C03630=1074.416,86.468,-68.167,173.484,24.240,154.290
C03631=1074.422,86.718,-68.185,173.486,24.243,154.290
C03632=1074.428,86.966,-68.204,173.487,24.245,154.290
C03633=1074.434,87.216,-68.222,173.489,24.248,154.290
C03634=1074.440,87.465,-68.239,173.491,24.251,154.291
C03635=1074.446,87.715,-68.257,173.492,24.253,154.291
C03636=1074.451,87.964,-68.275,173.493,24.256,154.291
C03637=1074.458,88.213,-68.293,173.496,24.259,154.292
C03638=1074.463,88.462,-68.311,173.497,24.261,154.292
C03639=1074.469,88.712,-68.329,173.498,24.263,154.292
C03640=1074.475,88.961,-68.346,173.500,24.266,154.293
C03641=1074.481,89.210,-68.366,173.502,24.269,154.293
C03642=1074.486,89.459,-68.383,173.503,24.271,154.293
C03643=1074.492,89.709,-68.401,173.504,24.274,154.294
C03644=1074.498,89.958,-68.419,173.506,24.276,154.294
C03645=1074.504,90.207,-68.437,173.508,24.279,154.294
C03646=1074.510,90.457,-68.455,173.509,24.282,154.294
C03647=1074.516,90.706,-68.473,173.511,24.284,154.295
C03648=1074.522,90.955,-68.491,173.512,24.286,154.295
C03649=1074.527,91.204,-68.510,173.514,24.289,154.295
C03650=1074.533,91.454,-68.528,173.516,24.292,154.296
C03651=1074.539,91.702,-68.546,173.517,24.294,154.296
C03652=1074.544,91.952,-68.564,173.519,24.297,154.296
C03653=1074.550,92.201,-68.582,173.521,24.299,154.297
C03654=1074.556,92.451,-68.601,173.522,24.302,154.297
C03655=1074.561,92.700,-68.619,173.523,24.305,154.297
C03656=1074.567,92.950,-68.637,173.525,24.307,154.298
C03657=1074.573,93.198,-68.655,173.527,24.310,154.298
C03658=1074.578,93.448,-68.673,173.528,24.313,154.298
C03659=1074.584,93.697,-68.692,173.529,24.315,154.299
C03660=1074.590,93.946,-68.710,173.532,24.318,154.299
C03661=1074.595,94.196,-68.728,173.533,24.321,154.299
C03662=1074.602,94.445,-68.747,173.534,24.323,154.299
C03663=1074.608,94.727,-68.768,173.536,24.326,154.300
C03664=1074.614,95.008,-68.788,173.538,24.329,154.300
C03665=1074.621,95.290,-68.808,173.540,24.332,154.301
C03666=1074.627,95.571,-68.829,173.541,24.334,154.301
C03667=1074.633,95.820,-68.848,173.543,24.337,154.301
C03668=1074.639,96.070,-68.866,173.545,24.340,154.301
C03669=1074.644,96.319,-68.884,173.546,24.342,154.302
C03670=1074.651,96.568,-68.902,173.547,24.344,154.302
C03671=1074.656,96.817,-68.921,173.549,24.348,154.302
C03672=1074.662,97.067,-68.939,173.551,24.350,154.303
C03673=1074.668,97.316,-68.958,173.552,24.352,154.303
C03674=1074.673,97.565,-68.976,173.555,24.355,154.303
C03675=1074.679,97.814,-68.995,173.556,24.358,154.304
C03676=1074.684,98.064,-69.013,173.557,24.360,154.304
C03677=1074.691,98.313,-69.031,173.558,24.363,154.304
C03678=1074.697,98.563,-69.049,173.561,24.365,154.304
C03679=1074.702,98.811,-69.068,173.562,24.368,154.305
C03680=1074.708,99.061,-69.087,173.563,24.370,154.305
C03681=1074.714,99.311,-69.105,173.566,24.373,154.305
C03682=1074.719,99.559,-69.124,173.567,24.376,154.306
C03683=1074.726,99.809,-69.142,173.568,24.378,154.306
C03684=1074.731,100.058,-69.161,173.570,24.381,154.306
C03685=1074.737,100.307,-69.179,173.572,24.383,154.307
C03686=1074.742,100.557,-69.198,173.573,24.386,154.307
C03687=1074.749,100.806,-69.216,173.575,24.388,154.307
C03688=1074.754,101.055,-69.235,173.577,24.391,154.308
C03689=1074.760,101.304,-69.253,173.578,24.394,154.308
C03690=1074.766,101.554,-69.272,173.580,24.396,154.308
C03691=1074.772,101.802,-69.291,173.581,24.398,154.308
C03692=1074.777,102.052,-69.309,173.583,24.401,154.309
C03693=1074.783,102.301,-69.327,173.584,24.404,154.309
C03694=1074.788,102.550,-69.347,173.586,24.406,154.309
C03695=1074.794,102.800,-69.365,173.588,24.409,154.310
C03696=1074.800,103.049,-69.384,173.589,24.412,154.310
C03697=1074.805,103.298,-69.403,173.591,24.414,154.310
C03698=1074.811,103.547,-69.422,173.593,24.417,154.311
C03699=1074.817,103.796,-69.440,173.594,24.419,154.311
C03700=1074.822,104.046,-69.459,173.596,24.422,154.311
C03701=1074.829,104.295,-69.477,173.597,24.424,154.312
C03702=1074.834,104.544,-69.496,173.599,24.427,154.312
C03703=1074.839,104.793,-69.516,173.601,24.429,154.312
C03704=1074.846,105.043,-69.534,173.602,24.432,154.312
C03705=1074.851,105.292,-69.552,173.604,24.435,154.313
C03706=1074.856,105.541,-69.572,173.606,24.437,154.313
C03707=1074.863,105.790,-69.590,173.607,24.440,154.313
C03708=1074.868,106.040,-69.610,173.609,24.442,154.314
C03709=1074.873,106.289,-69.628,173.611,24.445,154.314
C03710=1074.880,106.538,-69.646,173.612,24.447,154.314
C03711=1074.885,106.788,-69.666,173.614,24.450,154.315
C03712=1074.890,107.036,-69.684,173.615,24.453,154.315
C03713=1074.897,107.285,-69.703,173.617,24.455,154.315
C03714=1074.903,107.535,-69.722,173.618,24.457,154.315
C03715=1074.908,107.784,-69.742,173.620,24.460,154.316
C03716=1074.914,108.033,-69.760,173.622,24.463,154.316
C03717=1074.919,108.283,-69.778,173.623,24.465,154.316
C03718=1074.925,108.532,-69.798,173.625,24.468,154.317
C03719=1074.932,108.781,-69.816,173.627,24.470,154.317
C03720=1074.937,109.030,-69.835,173.628,24.473,154.317
C03721=1074.942,109.279,-69.854,173.630,24.476,154.317
C03722=1074.948,109.529,-69.874,173.632,24.478,154.318
C03723=1074.954,109.778,-69.892,173.633,24.480,154.318
C03724=1074.960,110.027,-69.912,173.635,24.483,154.318
C03725=1074.965,110.276,-69.930,173.637,24.486,154.319
C03726=1074.972,110.525,-69.949,173.638,24.488,154.319
C03727=1074.978,110.807,-69.971,173.640,24.491,154.319
C03728=1074.985,111.089,-69.992,173.642,24.494,154.320
C03729=1074.991,111.370,-70.014,173.644,24.496,154.320
C03730=1074.998,111.652,-70.036,173.646,24.500,154.320
C03731=1075.003,111.901,-70.055,173.647,24.502,154.321
C03732=1075.009,112.151,-70.074,173.650,24.505,154.321
C03733=1075.015,112.400,-70.093,173.651,24.507,154.321
C03734=1075.020,112.648,-70.112,173.652,24.509,154.321
C03735=1075.026,112.898,-70.131,173.655,24.513,154.322
C03736=1075.032,113.147,-70.150,173.656,24.515,154.322
C03737=1075.037,113.397,-70.169,173.657,24.517,154.322
C03738=1075.043,113.646,-70.189,173.660,24.520,154.323
C03739=1075.048,113.895,-70.207,173.661,24.522,154.323
C03740=1075.055,114.144,-70.226,173.662,24.525,154.323
C03741=1075.061,114.393,-70.246,173.665,24.527,154.323
C03742=1075.066,114.642,-70.265,173.666,24.530,154.324
C03743=1075.072,114.892,-70.285,173.667,24.533,154.324
C03744=1075.077,115.140,-70.303,173.670,24.535,154.324
C03745=1075.083,115.390,-70.323,173.671,24.538,154.325
C03746=1075.089,115.639,-70.342,173.672,24.541,154.325
C03747=1075.095,115.888,-70.362,173.675,24.543,154.325
C03748=1075.099,116.138,-70.382,173.676,24.546,154.326
C03749=1075.105,116.387,-70.401,173.677,24.548,154.326
C03750=1075.110,116.636,-70.420,173.680,24.551,154.326
C03751=1075.116,116.885,-70.439,173.681,24.554,154.327
C03752=1075.122,117.134,-70.459,173.682,24.556,154.327
C03753=1075.128,117.384,-70.478,173.684,24.559,154.327
C03754=1075.133,117.633,-70.498,173.686,24.561,154.327
C03755=1075.138,117.882,-70.516,173.687,24.563,154.328
C03756=1075.144,118.131,-70.536,173.689,24.566,154.328
C03757=1075.150,118.380,-70.556,173.691,24.569,154.328
C03758=1075.156,118.630,-70.575,173.693,24.572,154.329
C03759=1075.162,118.878,-70.595,173.694,24.574,154.329
C03760=1075.167,119.128,-70.614,173.696,24.576,154.329
C03761=1075.173,119.377,-70.633,173.698,24.579,154.330
C03762=1075.177,119.626,-70.653,173.699,24.582,154.330
C03763=1075.183,119.875,-70.673,173.701,24.584,154.330
C03764=1075.189,120.125,-70.692,173.703,24.587,154.330
C03765=1075.195,120.374,-70.711,173.704,24.589,154.331
C03766=1075.201,120.623,-70.731,173.707,24.592,154.331
C03767=1075.207,120.872,-70.750,173.708,24.594,154.331
C03768=1075.213,121.121,-70.770,173.710,24.597,154.332
C03769=1075.218,121.370,-70.790,173.712,24.600,154.332
C03770=1075.224,121.620,-70.809,173.713,24.602,154.332
C03771=1075.229,121.869,-70.829,173.714,24.604,154.333
C03772=1075.234,122.118,-70.848,173.717,24.607,154.333
C03773=1075.240,122.367,-70.868,173.718,24.609,154.333
C03774=1075.246,122.616,-70.887,173.720,24.612,154.333
C03775=1075.252,122.865,-70.907,173.722,24.614,154.334
C03776=1075.258,123.114,-70.927,173.723,24.617,154.334
C03777=1075.263,123.364,-70.946,173.726,24.619,154.334
C03778=1075.269,123.613,-70.966,173.727,24.622,154.335
C03779=1075.274,123.862,-70.986,173.728,24.625,154.335
C03780=1075.280,124.111,-71.006,173.730,24.627,154.335
C03781=1075.286,124.360,-71.025,173.732,24.630,154.335
C03782=1075.292,124.609,-71.045,173.734,24.632,154.336
C03783=1075.298,124.859,-71.064,173.736,24.635,154.336
C03784=1075.304,125.108,-71.084,173.737,24.637,154.336
C03785=1075.309,125.357,-71.104,173.739,24.640,154.337
C03786=1075.315,125.606,-71.124,173.741,24.642,154.337
C03787=1075.320,125.856,-71.143,173.743,24.645,154.337
C03788=1075.326,126.104,-71.163,173.744,24.647,154.337
C03789=1075.332,126.354,-71.182,173.746,24.649,154.338
C03790=1075.337,126.603,-71.203,173.748,24.652,154.338
C03791=1075.344,126.885,-71.225,173.750,24.655,154.338
C03792=1075.351,127.166,-71.247,173.752,24.658,154.339
C03793=1075.357,127.448,-71.270,173.754,24.661,154.339
C03794=1075.364,127.729,-71.292,173.756,24.664,154.339
C03795=1075.370,127.978,-71.312,173.757,24.666,154.340
C03796=1075.374,128.228,-71.332,173.760,24.669,154.340
C03797=1075.380,128.477,-71.352,173.761,24.671,154.340
C03798=1075.386,128.725,-71.371,173.762,24.673,154.340
C03799=1075.392,128.975,-71.391,173.765,24.676,154.341
C03800=1075.399,129.224,-71.411,173.766,24.678,154.341
C03801=1075.404,129.473,-71.432,173.768,24.681,154.341
C03802=1075.410,129.723,-71.451,173.770,24.683,154.341
C03803=1075.416,129.972,-71.471,173.771,24.686,154.342
C03804=1075.422,130.220,-71.491,173.774,24.688,154.342
C03805=1075.427,130.470,-71.511,173.775,24.691,154.342
C03806=1075.433,130.719,-71.531,173.777,24.693,154.343
C03807=1075.439,130.968,-71.551,173.779,24.696,154.343
C03808=1075.445,131.217,-71.570,173.781,24.698,154.343
C03809=1075.450,131.466,-71.590,173.782,24.701,154.343
C03810=1075.456,131.716,-71.611,173.784,24.703,154.344
C03811=1075.462,131.965,-71.631,173.786,24.706,154.344
C03812=1075.468,132.214,-71.651,173.787,24.708,154.344
C03813=1075.473,132.463,-71.671,173.790,24.711,154.345
C03814=1075.479,132.712,-71.690,173.791,24.713,154.345
C03815=1075.484,132.961,-71.711,173.793,24.716,154.345
C03816=1075.490,133.210,-71.731,173.795,24.718,154.345
C03817=1075.496,133.459,-71.751,173.796,24.720,154.346
C03818=1075.502,133.708,-71.771,173.799,24.723,154.346
C03819=1075.507,133.958,-71.791,173.800,24.725,154.346
C03820=1075.513,134.207,-71.811,173.802,24.729,154.347
C03821=1075.518,134.456,-71.832,173.804,24.731,154.347
C03822=1075.524,134.705,-71.852,173.806,24.734,154.347
C03823=1075.530,134.954,-71.873,173.807,24.736,154.347
C03824=1075.536,135.203,-71.893,173.810,24.739,154.348
C03825=1075.541,135.452,-71.913,173.811,24.741,154.348
C03826=1075.547,135.701,-71.933,173.812,24.743,154.348
C03827=1075.552,135.950,-71.954,173.815,24.746,154.349
C03828=1075.558,136.200,-71.973,173.816,24.748,154.349
C03829=1075.564,136.449,-71.994,173.818,24.751,154.349
C03830=1075.570,136.698,-72.014,173.820,24.753,154.349
C03831=1075.575,136.947,-72.034,173.822,24.756,154.350
C03832=1075.581,137.196,-72.054,173.823,24.758,154.350
C03833=1075.586,137.445,-72.075,173.826,24.761,154.350
C03834=1075.592,137.694,-72.095,173.827,24.763,154.350
C03835=1075.598,137.944,-72.116,173.829,24.766,154.351
C03836=1075.604,138.193,-72.136,173.831,24.768,154.351
C03837=1075.609,138.442,-72.156,173.832,24.771,154.351
C03838=1075.615,138.691,-72.176,173.835,24.773,154.352
C03839=1075.621,138.940,-72.197,173.836,24.776,154.352
C03840=1075.626,139.189,-72.217,173.838,24.778,154.352
C03841=1075.632,139.438,-72.238,173.840,24.781,154.352
C03842=1075.638,139.688,-72.258,173.842,24.783,154.353
C03843=1075.644,139.936,-72.278,173.843,24.786,154.353
C03844=1075.649,140.185,-72.299,173.846,24.788,154.353
C03845=1075.654,140.434,-72.320,173.847,24.791,154.353
C03846=1075.661,140.684,-72.340,173.849,24.793,154.354
C03847=1075.666,140.933,-72.361,173.851,24.796,154.354
C03848=1075.672,141.182,-72.381,173.853,24.798,154.354
C03849=1075.678,141.431,-72.401,173.855,24.801,154.355
C03850=1075.683,141.680,-72.422,173.857,24.803,154.355
C03851=1075.689,141.930,-72.443,173.858,24.806,154.355
C03852=1075.694,142.178,-72.464,173.861,24.808,154.355
C03853=1075.700,142.427,-72.484,173.862,24.811,154.356
C03854=1075.705,142.676,-72.505,173.864,24.813,154.356
C03855=1075.712,142.958,-72.528,173.866,24.816,154.356
C03856=1075.719,143.239,-72.551,173.868,24.819,154.357
C03857=1075.725,143.520,-72.574,173.870,24.822,154.357
C03858=1075.731,143.802,-72.598,173.872,24.825,154.357
C03859=1075.736,144.051,-72.618,173.874,24.827,154.358
C03860=1075.742,144.301,-72.639,173.876,24.830,154.358
C03861=1075.748,144.549,-72.661,173.878,24.832,154.358
C03862=1075.754,144.798,-72.680,173.880,24.835,154.358
C03863=1075.759,145.047,-72.701,173.881,24.837,154.359
C03864=1075.765,145.297,-72.722,173.884,24.840,154.359
C03865=1075.770,145.546,-72.743,173.885,24.842,154.359
C03866=1075.776,145.795,-72.763,173.887,24.845,154.359
C03867=1075.782,146.044,-72.784,173.889,24.847,154.360
C03868=1075.788,146.293,-72.805,173.891,24.850,154.360
C03869=1075.793,146.542,-72.826,173.892,24.852,154.360
C03870=1075.799,146.791,-72.846,173.895,24.855,154.361
C03871=1075.805,147.040,-72.868,173.896,24.857,154.361
C03872=1075.811,147.289,-72.888,173.898,24.860,154.361
C03873=1075.816,147.538,-72.909,173.900,24.862,154.361
C03874=1075.822,147.787,-72.930,173.902,24.865,154.362
C03875=1075.828,148.036,-72.950,173.904,24.867,154.362
C03876=1075.833,148.285,-72.971,173.906,24.870,154.362
C03877=1075.839,148.535,-72.992,173.908,24.872,154.362
C03878=1075.845,148.784,-73.013,173.910,24.875,154.363
C03879=1075.850,149.032,-73.034,173.912,24.877,154.363
C03880=1075.856,149.282,-73.055,173.913,24.880,154.363
C03881=1075.862,149.531,-73.076,173.916,24.882,154.364
C03882=1075.867,149.780,-73.097,173.917,24.885,154.364
C03883=1075.873,150.030,-73.118,173.919,24.887,154.364
C03884=1075.878,150.278,-73.139,173.921,24.890,154.364
C03885=1075.884,150.527,-73.160,173.923,24.892,154.365
C03886=1075.890,150.776,-73.181,173.925,24.895,154.365
C03887=1075.895,151.025,-73.202,173.927,24.897,154.365
C03888=1075.901,151.274,-73.223,173.928,24.899,154.366
C03889=1075.906,151.524,-73.244,173.931,24.902,154.366
C03890=1075.912,151.772,-73.265,173.932,24.904,154.366
C03891=1075.917,152.021,-73.286,173.934,24.907,154.366
C03892=1075.923,152.271,-73.308,173.937,24.910,154.367
C03893=1075.929,152.519,-73.329,173.938,24.912,154.367
C03894=1075.935,152.769,-73.350,173.940,24.915,154.367
C03895=1075.940,153.017,-73.371,173.942,24.917,154.367
C03896=1075.946,153.267,-73.392,173.944,24.920,154.368
C03897=1075.952,153.516,-73.413,173.946,24.922,154.368
C03898=1075.957,153.765,-73.434,173.948,24.924,154.368
C03899=1075.963,154.013,-73.455,173.949,24.926,154.368
C03900=1075.969,154.263,-73.477,173.952,24.929,154.369
C03901=1075.974,154.512,-73.497,173.954,24.932,154.369
C03902=1075.980,154.761,-73.519,173.956,24.934,154.369
C03903=1075.986,155.009,-73.540,173.958,24.937,154.369
C03904=1075.992,155.259,-73.561,173.959,24.939,154.370
C03905=1075.997,155.508,-73.582,173.962,24.942,154.370
C03906=1076.003,155.756,-73.604,173.963,24.944,154.370
C03907=1076.009,156.006,-73.625,173.965,24.947,154.371
C03908=1076.013,156.255,-73.646,173.968,24.949,154.371
C03909=1076.020,156.504,-73.668,173.969,24.952,154.371
C03910=1076.025,156.753,-73.689,173.971,24.954,154.371
C03911=1076.031,157.002,-73.710,173.973,24.957,154.372
C03912=1076.037,157.251,-73.731,173.975,24.959,154.372
C03913=1076.042,157.499,-73.753,173.977,24.962,154.372
C03914=1076.047,157.750,-73.774,173.979,24.964,154.373
C03915=1076.053,157.998,-73.796,173.981,24.967,154.373
C03916=1076.059,158.247,-73.817,173.983,24.969,154.373
C03917=1076.064,158.496,-73.838,173.985,24.972,154.373
C03918=1076.071,158.745,-73.860,173.986,24.974,154.374
C03919=1076.076,159.027,-73.884,173.989,24.977,154.374
C03920=1076.083,159.307,-73.908,173.991,24.980,154.374
C03921=1076.089,159.589,-73.932,173.993,24.983,154.375
C03922=1076.096,159.870,-73.957,173.996,24.985,154.375
C03923=1076.102,160.119,-73.978,173.998,24.988,154.375
C03924=1076.107,160.368,-74.000,173.999,24.990,154.375
C03925=1076.113,160.618,-74.021,174.002,24.993,154.376
C03926=1076.118,160.866,-74.042,174.003,24.995,154.376
C03927=1076.124,161.115,-74.064,174.005,24.998,154.376
C03928=1076.129,161.364,-74.086,174.008,25.001,154.376
C03929=1076.135,161.613,-74.107,174.009,25.003,154.377
C03930=1076.141,161.862,-74.129,174.011,25.006,154.377
C03931=1076.146,162.111,-74.151,174.013,25.008,154.377
C03932=1076.152,162.360,-74.172,174.015,25.011,154.378
C03933=1076.157,162.609,-74.194,174.018,25.013,154.378
C03934=1076.163,162.858,-74.216,174.019,25.016,154.378
C03935=1076.168,163.107,-74.238,174.021,25.018,154.378
C03936=1076.174,163.356,-74.259,174.024,25.021,154.379
C03937=1076.179,163.605,-74.281,174.025,25.024,154.379
C03938=1076.185,163.854,-74.303,174.027,25.026,154.379
C03939=1076.190,164.103,-74.325,174.029,25.029,154.380
C03940=1076.195,164.352,-74.347,174.031,25.031,154.380
C03941=1076.201,164.601,-74.368,174.033,25.034,154.380
C03942=1076.206,164.850,-74.390,174.035,25.036,154.380
C03943=1076.212,165.099,-74.412,174.037,25.039,154.381
C03944=1076.217,165.348,-74.434,174.039,25.042,154.381
C03945=1076.223,165.597,-74.455,174.041,25.044,154.381
C03946=1076.228,165.846,-74.477,174.043,25.047,154.381
C03947=1076.234,166.095,-74.499,174.045,25.049,154.382
C03948=1076.239,166.344,-74.521,174.047,25.051,154.382
C03949=1076.245,166.593,-74.543,174.049,25.054,154.382
C03950=1076.250,166.842,-74.565,174.051,25.056,154.383
C03951=1076.256,167.091,-74.587,174.053,25.059,154.383
C03952=1076.261,167.340,-74.608,174.055,25.062,154.383
C03953=1076.267,167.589,-74.631,174.057,25.064,154.383
C03954=1076.272,167.838,-74.652,174.059,25.067,154.384
C03955=1076.278,168.087,-74.675,174.061,25.069,154.384
C03956=1076.284,168.335,-74.696,174.063,25.072,154.384
C03957=1076.289,168.585,-74.718,174.065,25.075,154.385
C03958=1076.294,168.834,-74.741,174.067,25.077,154.385
C03959=1076.300,169.083,-74.762,174.069,25.080,154.385
C03960=1076.306,169.332,-74.785,174.071,25.082,154.385
C03961=1076.311,169.580,-74.806,174.074,25.085,154.386
C03962=1076.317,169.830,-74.828,174.075,25.087,154.386
C03963=1076.322,170.079,-74.851,174.077,25.090,154.386
C03964=1076.328,170.327,-74.873,174.080,25.093,154.386
C03965=1076.333,170.577,-74.895,174.081,25.095,154.387
C03966=1076.340,170.826,-74.916,174.083,25.098,154.387
C03967=1076.344,171.075,-74.938,174.086,25.100,154.387
C03968=1076.350,171.324,-74.961,174.087,25.102,154.387
C03969=1076.356,171.573,-74.983,174.090,25.105,154.388
C03970=1076.361,171.822,-75.005,174.092,25.107,154.388
C03971=1076.368,172.070,-75.027,174.093,25.110,154.388
C03972=1076.373,172.320,-75.049,174.096,25.112,154.389
C03973=1076.378,172.568,-75.072,174.098,25.115,154.389
C03974=1076.384,172.817,-75.094,174.100,25.117,154.389
C03975=1076.390,173.067,-75.116,174.102,25.120,154.389
C03976=1076.395,173.315,-75.138,174.104,25.122,154.390
C03977=1076.401,173.564,-75.160,174.106,25.125,154.390
C03978=1076.407,173.813,-75.183,174.108,25.127,154.390
C03979=1076.412,174.062,-75.205,174.110,25.130,154.390
C03980=1076.418,174.311,-75.226,174.113,25.133,154.391
C03981=1076.423,174.560,-75.249,174.114,25.135,154.391
C03982=1076.429,174.809,-75.272,174.116,25.138,154.391
C03983=1076.435,175.090,-75.297,174.119,25.140,154.392
C03984=1076.441,175.370,-75.322,174.121,25.143,154.392
C03985=1076.448,175.651,-75.346,174.123,25.146,154.392
C03986=1076.454,175.932,-75.372,174.126,25.149,154.392
C03987=1076.460,176.181,-75.395,174.128,25.151,154.393
C03988=1076.466,176.430,-75.417,174.130,25.154,154.393
C03989=1076.472,176.679,-75.439,174.132,25.156,154.393
C03990=1076.478,176.928,-75.461,174.134,25.159,154.394
C03991=1076.483,177.177,-75.484,174.137,25.162,154.394
C03992=1076.488,177.426,-75.506,174.139,25.164,154.394
C03993=1076.495,177.675,-75.529,174.140,25.167,154.394
C03994=1076.500,177.924,-75.551,174.143,25.169,154.394
C03995=1076.506,178.173,-75.574,174.145,25.171,154.395
C03996=1076.512,178.421,-75.596,174.147,25.174,154.395
C03997=1076.517,178.671,-75.618,174.149,25.176,154.395
C03998=1076.523,178.919,-75.641,174.151,25.179,154.396
C03999=1076.528,179.168,-75.664,174.154,25.181,154.396
C04000=1076.535,179.418,-75.685,174.155,25.184,154.396
C04001=1076.540,179.666,-75.708,174.157,25.186,154.396
C04002=1076.545,179.915,-75.731,174.160,25.189,154.397
C04003=1076.551,180.164,-75.753,174.162,25.191,154.397
C04004=1076.557,180.413,-75.776,174.164,25.193,154.397
C04005=1076.563,180.662,-75.798,174.166,25.196,154.397
C04006=1076.569,180.911,-75.821,174.168,25.199,154.398
C04007=1076.574,181.160,-75.844,174.171,25.201,154.398
C04008=1076.581,181.409,-75.866,174.172,25.204,154.398
C04009=1076.586,181.657,-75.889,174.174,25.206,154.398
C04010=1076.591,181.906,-75.911,174.177,25.209,154.399
C04011=1076.597,182.155,-75.934,174.179,25.211,154.399
C04012=1076.603,182.404,-75.956,174.181,25.213,154.399
C04013=1076.609,182.653,-75.979,174.183,25.216,154.399
C04014=1076.615,182.902,-76.001,174.185,25.219,154.400
C04015=1076.620,183.151,-76.024,174.188,25.221,154.400
C04016=1076.626,183.400,-76.047,174.190,25.224,154.400
C04017=1076.633,183.649,-76.070,174.192,25.226,154.400
C04018=1076.638,183.897,-76.092,174.194,25.228,154.401
C04019=1076.644,184.147,-76.115,174.196,25.231,154.401
C04020=1076.649,184.396,-76.138,174.199,25.233,154.401
C04021=1076.655,184.645,-76.161,174.200,25.236,154.401
C04022=1076.662,184.893,-76.183,174.203,25.238,154.402
C04023=1076.666,185.142,-76.206,174.205,25.241,154.402
C04024=1076.672,185.391,-76.229,174.207,25.244,154.402
C04025=1076.678,185.640,-76.252,174.210,25.246,154.402
C04026=1076.683,185.889,-76.275,174.211,25.249,154.403
C04027=1076.689,186.137,-76.298,174.213,25.251,154.403
C04028=1076.694,186.387,-76.321,174.216,25.254,154.403
C04029=1076.700,186.636,-76.344,174.218,25.256,154.404
C04030=1076.705,186.884,-76.367,174.220,25.259,154.404
C04031=1076.711,187.133,-76.390,174.222,25.261,154.404
C04032=1076.716,187.382,-76.413,174.224,25.265,154.405
C04033=1076.721,187.631,-76.436,174.226,25.267,154.405
C04034=1076.727,187.880,-76.459,174.229,25.270,154.405
C04035=1076.733,188.129,-76.482,174.231,25.272,154.405
C04036=1076.738,188.377,-76.505,174.233,25.275,154.406
C04037=1076.743,188.627,-76.529,174.235,25.277,154.406
C04038=1076.749,188.876,-76.552,174.237,25.280,154.406
C04039=1076.755,189.124,-76.575,174.240,25.283,154.406
C04040=1076.760,189.373,-76.597,174.242,25.285,154.407
C04041=1076.765,189.622,-76.621,174.244,25.288,154.407
C04042=1076.771,189.871,-76.644,174.246,25.290,154.407
C04043=1076.777,190.120,-76.667,174.248,25.293,154.407
C04044=1076.782,190.369,-76.690,174.251,25.295,154.408
C04045=1076.787,190.618,-76.713,174.253,25.298,154.408
C04046=1076.793,190.866,-76.737,174.255,25.301,154.408
C04047=1076.800,191.147,-76.762,174.258,25.304,154.409
C04048=1076.806,191.427,-76.789,174.260,25.306,154.409
C04049=1076.812,191.707,-76.815,174.262,25.310,154.409
C04050=1076.818,191.988,-76.841,174.264,25.312,154.410
C04051=1076.824,192.237,-76.864,174.267,25.315,154.410
C04052=1076.830,192.486,-76.888,174.269,25.317,154.410
C04053=1076.835,192.735,-76.911,174.272,25.320,154.410
C04054=1076.841,192.984,-76.934,174.274,25.323,154.411
C04055=1076.846,193.233,-76.957,174.276,25.325,154.411
C04056=1076.852,193.481,-76.981,174.278,25.328,154.411
C04057=1076.857,193.730,-77.004,174.280,25.330,154.411
C04058=1076.863,193.979,-77.027,174.282,25.333,154.412
C04059=1076.868,194.228,-77.051,174.285,25.336,154.412
C04060=1076.874,194.476,-77.075,174.287,25.338,154.412
C04061=1076.880,194.725,-77.097,174.290,25.341,154.413
C04062=1076.886,194.975,-77.121,174.292,25.343,154.413
C04063=1076.892,195.224,-77.145,174.293,25.346,154.413
C04064=1076.897,195.472,-77.168,174.296,25.349,154.413
C04065=1076.903,195.721,-77.191,174.298,25.351,154.414
C04066=1076.908,195.970,-77.215,174.300,25.354,154.414
C04067=1076.914,196.219,-77.238,174.303,25.357,154.414
C04068=1076.919,196.467,-77.262,174.305,25.359,154.415
C04069=1076.925,196.716,-77.285,174.307,25.362,154.415
C04070=1076.931,196.965,-77.308,174.310,25.365,154.415
C04071=1076.936,197.214,-77.333,174.312,25.367,154.415
C04072=1076.942,197.463,-77.355,174.314,25.369,154.416
C04073=1076.948,197.712,-77.380,174.316,25.372,154.416
C04074=1076.953,197.961,-77.403,174.318,25.375,154.416
C04075=1076.959,198.209,-77.427,174.321,25.377,154.416
C04076=1076.965,198.458,-77.450,174.323,25.380,154.417
C04077=1076.971,198.707,-77.474,174.325,25.383,154.417
C04078=1076.976,198.955,-77.497,174.328,25.385,154.417
C04079=1076.982,199.205,-77.521,174.330,25.388,154.418
C04080=1076.988,199.454,-77.544,174.332,25.390,154.418
C04081=1076.994,199.702,-77.568,174.335,25.393,154.418
C04082=1076.999,199.951,-77.592,174.336,25.395,154.418
C04083=1077.005,200.199,-77.615,174.339,25.397,154.418
C04084=1077.010,200.449,-77.639,174.341,25.400,154.419
C04085=1077.017,200.698,-77.663,174.343,25.403,154.419
C04086=1077.023,200.946,-77.687,174.346,25.405,154.419
C04087=1077.028,201.195,-77.710,174.348,25.408,154.420
C04088=1077.034,201.443,-77.734,174.351,25.410,154.420
C04089=1077.039,201.693,-77.758,174.353,25.413,154.420
C04090=1077.045,201.942,-77.781,174.355,25.416,154.420
C04091=1077.051,202.190,-77.806,174.358,25.418,154.421
C04092=1077.056,202.439,-77.828,174.360,25.421,154.421
C04093=1077.062,202.688,-77.853,174.362,25.424,154.421
C04094=1077.068,202.937,-77.877,174.365,25.427,154.422
C04095=1077.073,203.186,-77.900,174.367,25.429,154.422
C04096=1077.079,203.434,-77.925,174.368,25.432,154.422
C04097=1077.085,203.683,-77.948,174.371,25.434,154.422
C04098=1077.090,203.931,-77.972,174.373,25.437,154.423
C04099=1077.095,204.181,-77.996,174.376,25.439,154.423
C04100=1077.102,204.429,-78.020,174.378,25.442,154.423
C04101=1077.107,204.678,-78.044,174.380,25.445,154.423
C04102=1077.112,204.927,-78.069,174.383,25.448,154.424
C04103=1077.118,205.176,-78.092,174.385,25.450,154.424
C04104=1077.124,205.425,-78.116,174.387,25.453,154.424
C04105=1077.129,205.673,-78.140,174.390,25.456,154.425
C04106=1077.135,205.922,-78.164,174.392,25.458,154.425
C04107=1077.140,206.170,-78.188,174.394,25.461,154.425
C04108=1077.146,206.420,-78.212,174.397,25.463,154.425
C04109=1077.151,206.669,-78.236,174.399,25.466,154.426
C04110=1077.157,206.917,-78.260,174.402,25.469,154.426
C04111=1077.181,207.954,-78.361,174.513,25.528,154.425
C04112=1077.190,208.361,-78.401,174.516,25.534,154.426
C04113=1077.200,208.767,-78.442,174.520,25.540,154.427
C04114=1077.209,209.173,-78.482,174.524,25.546,154.428
C04115=1077.218,209.580,-78.523,174.527,25.552,154.429
C04116=1077.224,209.829,-78.548,174.529,25.555,154.429
C04117=1077.230,210.077,-78.573,174.532,25.558,154.430
C04118=1077.236,210.326,-78.597,174.534,25.562,154.430
C04119=1077.241,210.574,-78.622,174.536,25.566,154.431
C04120=1077.247,210.823,-78.647,174.538,25.569,154.431
C04121=1077.252,211.072,-78.671,174.540,25.573,154.432
C04122=1077.259,211.321,-78.696,174.542,25.577,154.432
C04123=1077.264,211.569,-78.721,174.544,25.580,154.433
C04124=1077.270,211.818,-78.746,174.546,25.584,154.433
C04125=1077.276,212.067,-78.771,174.549,25.587,154.434
C04126=1077.282,212.315,-78.796,174.551,25.591,154.434
C04127=1077.288,212.564,-78.821,174.553,25.594,154.435
C04128=1077.292,212.813,-78.846,174.555,25.598,154.435
C04129=1077.299,213.061,-78.871,174.558,25.602,154.436
C04130=1077.305,213.311,-78.896,174.560,25.606,154.436
C04131=1077.310,213.559,-78.921,174.562,25.609,154.437
C04132=1077.316,213.807,-78.946,174.564,25.613,154.437
C04133=1077.321,214.056,-78.971,174.567,25.616,154.438
C04134=1077.327,214.305,-78.996,174.569,25.620,154.438
C04135=1077.333,214.554,-79.021,174.571,25.624,154.439
C04136=1077.339,214.802,-79.046,174.573,25.627,154.439
C04137=1077.344,215.051,-79.072,174.575,25.631,154.440
C04138=1077.349,215.300,-79.096,174.577,25.634,154.440
C04139=1077.356,215.548,-79.121,174.579,25.638,154.441
C04140=1077.362,215.797,-79.147,174.582,25.642,154.441
C04141=1077.367,216.045,-79.172,174.585,25.646,154.442
C04142=1077.373,216.295,-79.197,174.587,25.649,154.442
C04143=1077.379,216.543,-79.222,174.589,25.652,154.443
C04144=1077.384,216.792,-79.248,174.591,25.656,154.443
C04145=1077.390,217.040,-79.273,174.593,25.660,154.444
C04146=1077.396,217.290,-79.298,174.595,25.663,154.444
C04147=1077.401,217.538,-79.323,174.597,25.667,154.445
C04148=1077.407,217.787,-79.349,174.600,25.671,154.445
C04149=1077.413,218.035,-79.374,174.602,25.674,154.446
C04150=1077.419,218.283,-79.399,174.605,25.678,154.446
C04151=1077.424,218.532,-79.425,174.607,25.681,154.447
C04152=1077.430,218.781,-79.449,174.609,25.685,154.447
C04153=1077.436,219.030,-79.475,174.611,25.689,154.448
C04154=1077.441,219.278,-79.500,174.613,25.692,154.448
C04155=1077.447,219.527,-79.526,174.616,25.696,154.449
C04156=1077.453,219.776,-79.551,174.618,25.699,154.449
C04157=1077.459,220.025,-79.577,174.620,25.703,154.450
C04158=1077.465,220.273,-79.602,174.622,25.706,154.450
C04159=1077.471,220.521,-79.627,174.625,25.710,154.451
C04160=1077.476,220.770,-79.653,174.627,25.714,154.451
C04161=1077.482,221.019,-79.679,174.630,25.717,154.452
C04162=1077.489,221.268,-79.704,174.632,25.721,154.452
C04163=1077.493,221.516,-79.729,174.634,25.724,154.453
C04164=1077.503,221.927,-79.772,174.637,25.730,154.454
C04165=1077.512,222.338,-79.814,174.641,25.736,154.454
C04166=1077.522,222.749,-79.856,174.646,25.742,154.455
C04167=1077.532,223.159,-79.899,174.649,25.748,154.456
C04168=1077.537,223.408,-79.924,174.651,25.752,154.457
C04169=1077.543,223.656,-79.949,174.653,25.756,154.457
C04170=1077.548,223.905,-79.975,174.656,25.759,154.458
C04171=1077.554,224.153,-80.001,174.658,25.763,154.458
C04172=1077.560,224.402,-80.027,174.661,25.767,154.459
C04173=1077.565,224.651,-80.053,174.663,25.770,154.459
C04174=1077.572,224.900,-80.078,174.665,25.774,154.460
C04175=1077.577,225.147,-80.104,174.667,25.777,154.460
C04176=1077.582,225.396,-80.130,174.669,25.781,154.461
C04177=1077.588,225.645,-80.155,174.672,25.784,154.461
C04178=1077.594,225.894,-80.181,174.674,25.788,154.462
C04179=1077.600,226.143,-80.207,174.677,25.792,154.462
C04180=1077.606,226.391,-80.233,174.679,25.795,154.463
C04181=1077.611,226.639,-80.259,174.681,25.799,154.463
C04182=1077.617,226.888,-80.284,174.683,25.802,154.464
C04183=1077.622,227.137,-80.310,174.686,25.806,154.464
C04184=1077.629,227.385,-80.336,174.688,25.810,154.465
C04185=1077.634,227.634,-80.362,174.691,25.814,154.465
C04186=1077.640,227.883,-80.388,174.693,25.817,154.466
C04187=1077.646,228.131,-80.414,174.695,25.820,154.466
C04188=1077.652,228.380,-80.440,174.697,25.824,154.467
C04189=1077.657,228.629,-80.466,174.699,25.828,154.467
C04190=1077.664,228.877,-80.492,174.703,25.832,154.468
C04191=1077.669,229.126,-80.518,174.705,25.835,154.468
C04192=1077.674,229.374,-80.544,174.707,25.838,154.469
C04193=1077.681,229.622,-80.570,174.709,25.842,154.469
C04194=1077.686,229.871,-80.596,174.711,25.846,154.470
C04195=1077.692,230.120,-80.622,174.714,25.849,154.470
C04196=1077.697,230.369,-80.648,174.717,25.853,154.471
C04197=1077.704,230.617,-80.674,174.719,25.856,154.471
C04198=1077.709,230.866,-80.700,174.721,25.860,154.472
C04199=1077.715,231.114,-80.727,174.723,25.863,154.472
C04200=1077.721,231.363,-80.753,174.725,25.867,154.473
C04201=1077.726,231.611,-80.779,174.728,25.871,154.473
C04202=1077.732,231.860,-80.805,174.730,25.875,154.474
C04203=1077.738,232.109,-80.831,174.733,25.878,154.474
C04204=1077.744,232.357,-80.857,174.735,25.881,154.475
C04205=1077.750,232.606,-80.884,174.737,25.885,154.475
C04206=1077.755,232.855,-80.910,174.740,25.889,154.476
C04207=1077.761,233.103,-80.937,174.742,25.893,154.476
C04208=1077.767,233.352,-80.963,174.744,25.896,154.477
C04209=1077.772,233.601,-80.989,174.747,25.900,154.477
C04210=1077.778,233.849,-81.016,174.749,25.903,154.478
C04211=1077.783,234.098,-81.042,174.752,25.907,154.478
C04212=1077.790,234.346,-81.068,174.754,25.910,154.479
C04213=1077.796,234.594,-81.094,174.756,25.914,154.479
C04214=1077.801,234.843,-81.120,174.758,25.918,154.480
C04215=1077.807,235.092,-81.147,174.762,25.922,154.480
C04216=1077.815,235.494,-81.190,174.765,25.928,154.481
C04217=1077.825,235.896,-81.233,174.769,25.933,154.482
C04218=1077.834,236.298,-81.275,174.773,25.939,154.483
C04219=1077.844,236.700,-81.319,174.776,25.945,154.483
C04220=1077.849,236.949,-81.345,174.779,25.948,154.484
C04221=1077.855,237.198,-81.372,174.782,25.952,154.484
C04222=1077.861,237.446,-81.398,174.784,25.956,154.485
C04223=1077.866,237.694,-81.425,174.786,25.959,154.485
C04224=1077.872,237.943,-81.452,174.789,25.963,154.486
C04225=1077.878,238.192,-81.477,174.791,25.966,154.486
C04226=1077.884,238.441,-81.504,174.793,25.970,154.487
C04227=1077.890,238.689,-81.531,174.796,25.974,154.487
C04228=1077.896,238.937,-81.558,174.799,25.977,154.488
C04229=1077.901,239.186,-81.584,174.801,25.981,154.488
C04230=1077.907,239.434,-81.611,174.803,25.985,154.489
C04231=1077.912,239.683,-81.638,174.805,25.988,154.489
C04232=1077.918,239.931,-81.665,174.808,25.992,154.490
C04233=1077.924,240.179,-81.692,174.811,25.995,154.490
C04234=1077.930,240.429,-81.719,174.813,25.999,154.491
C04235=1077.936,240.677,-81.745,174.815,26.003,154.491
C04236=1077.942,240.925,-81.772,174.818,26.006,154.492
C04237=1077.947,241.174,-81.799,174.820,26.010,154.492
C04238=1077.953,241.422,-81.825,174.822,26.013,154.493
C04239=1077.958,241.671,-81.852,174.825,26.017,154.493
C04240=1077.965,241.920,-81.879,174.828,26.021,154.494
C04241=1077.970,242.168,-81.906,174.830,26.024,154.494
C04242=1077.976,242.416,-81.933,174.832,26.028,154.495
C04243=1077.982,242.665,-81.959,174.834,26.031,154.495
C04244=1077.988,242.913,-81.986,174.837,26.035,154.496
C04245=1077.993,243.163,-82.014,174.840,26.039,154.496
C04246=1077.999,243.411,-82.040,174.842,26.042,154.497
C04247=1078.005,243.659,-82.067,174.845,26.046,154.497
C04248=1078.010,243.907,-82.095,174.847,26.050,154.498
C04249=1078.016,244.156,-82.122,174.849,26.053,154.498
C04250=1078.022,244.404,-82.148,174.851,26.057,154.499
C04251=1078.027,244.653,-82.176,174.855,26.061,154.499
C04252=1078.033,244.902,-82.202,174.857,26.064,154.500
C04253=1078.039,245.149,-82.230,174.859,26.067,154.500
C04254=1078.044,245.398,-82.257,174.862,26.071,154.501
C04255=1078.051,245.647,-82.284,174.864,26.075,154.501
C04256=1078.056,245.896,-82.311,174.867,26.079,154.502
C04257=1078.062,246.144,-82.339,174.869,26.082,154.503
C04258=1078.068,246.392,-82.365,174.872,26.086,154.503
C04259=1078.073,246.640,-82.392,174.874,26.090,154.504
C04260=1078.079,246.890,-82.420,174.876,26.093,154.504
C04261=1078.085,247.137,-82.447,174.879,26.097,154.505
C04262=1078.090,247.386,-82.474,174.881,26.101,154.505
C04263=1078.096,247.634,-82.501,174.884,26.104,154.506
C04264=1078.102,247.883,-82.529,174.887,26.108,154.506
C04265=1078.107,248.132,-82.556,174.889,26.112,154.507
C04266=1078.113,248.380,-82.584,174.891,26.116,154.507
C04267=1078.118,248.628,-82.611,174.893,26.119,154.508
C04268=1078.127,249.024,-82.655,174.898,26.125,154.508
C04269=1078.136,249.419,-82.698,174.902,26.131,154.509
C04270=1078.145,249.815,-82.741,174.905,26.136,154.510
C04271=1078.155,250.211,-82.785,174.910,26.142,154.511
C04272=1078.160,250.459,-82.813,174.912,26.146,154.511
C04273=1078.166,250.708,-82.841,174.914,26.150,154.512
C04274=1078.172,250.956,-82.868,174.917,26.154,154.512
C04275=1078.177,251.204,-82.895,174.920,26.157,154.513
C04276=1078.183,251.453,-82.924,174.922,26.161,154.514
C04277=1078.189,251.701,-82.951,174.924,26.164,154.514
C04278=1078.194,251.950,-82.978,174.927,26.168,154.515
C04279=1078.200,252.198,-83.006,174.929,26.172,154.515
C04280=1078.206,252.447,-83.033,174.932,26.176,154.516
C04281=1078.211,252.695,-83.061,174.935,26.179,154.516
C04282=1078.218,252.943,-83.089,174.937,26.183,154.517
C04283=1078.223,253.192,-83.116,174.940,26.187,154.517
C04284=1078.228,253.440,-83.144,174.942,26.190,154.518
C04285=1078.235,253.688,-83.172,174.944,26.194,154.518
C04286=1078.240,253.937,-83.199,174.948,26.197,154.519
C04287=1078.246,254.186,-83.227,174.950,26.201,154.519
C04288=1078.252,254.434,-83.255,174.952,26.205,154.520
C04289=1078.257,254.682,-83.283,174.955,26.208,154.520
C04290=1078.263,254.931,-83.310,174.957,26.212,154.521
C04291=1078.269,255.179,-83.338,174.960,26.216,154.521
C04292=1078.275,255.427,-83.366,174.963,26.220,154.522
C04293=1078.280,255.675,-83.394,174.965,26.223,154.522
C04294=1078.286,255.925,-83.421,174.967,26.227,154.523
C04295=1078.292,256.173,-83.449,174.970,26.231,154.523
C04296=1078.298,256.421,-83.477,174.972,26.234,154.524
C04297=1078.304,256.669,-83.505,174.975,26.238,154.524
C04298=1078.309,256.917,-83.533,174.978,26.241,154.525
C04299=1078.315,257.166,-83.561,174.980,26.245,154.525
C04300=1078.320,257.415,-83.588,174.983,26.249,154.526
C04301=1078.327,257.663,-83.616,174.985,26.252,154.526
C04302=1078.332,257.911,-83.644,174.988,26.256,154.527
C04303=1078.338,258.160,-83.672,174.991,26.260,154.527
C04304=1078.344,258.409,-83.700,174.993,26.263,154.528
C04305=1078.350,258.656,-83.728,174.996,26.267,154.528
C04306=1078.356,258.905,-83.756,174.998,26.271,154.529
C04307=1078.361,259.153,-83.784,175.001,26.274,154.529
C04308=1078.367,259.402,-83.812,175.004,26.278,154.530
C04309=1078.373,259.650,-83.840,175.006,26.281,154.530
C04310=1078.379,259.898,-83.868,175.008,26.285,154.531
C04311=1078.385,260.146,-83.896,175.011,26.289,154.531
C04312=1078.391,260.395,-83.924,175.013,26.292,154.532
C04313=1078.397,260.644,-83.952,175.017,26.296,154.532
C04314=1078.403,260.892,-83.980,175.019,26.300,154.533
C04315=1078.409,261.140,-84.008,175.021,26.303,154.533
C04316=1078.414,261.388,-84.036,175.024,26.307,154.534
C04317=1078.420,261.637,-84.065,175.026,26.310,154.534
C04318=1078.427,261.885,-84.093,175.030,26.314,154.535
C04319=1078.432,262.133,-84.121,175.032,26.318,154.535
C04320=1078.441,262.526,-84.166,175.035,26.323,154.536
C04321=1078.451,262.919,-84.210,175.040,26.329,154.537
C04322=1078.460,263.312,-84.255,175.044,26.335,154.538
C04323=1078.470,263.705,-84.300,175.049,26.341,154.539
C04324=1078.475,263.953,-84.328,175.051,26.344,154.539
C04325=1078.481,264.201,-84.357,175.054,26.348,154.539
C04326=1078.487,264.450,-84.385,175.056,26.351,154.540
C04327=1078.493,264.698,-84.413,175.058,26.356,154.541
C04328=1078.499,264.946,-84.442,175.062,26.359,154.541
C04329=1078.504,265.194,-84.470,175.064,26.363,154.542
C04330=1078.510,265.443,-84.499,175.067,26.367,154.542
C04331=1078.516,265.691,-84.528,175.069,26.370,154.543
C04332=1078.522,265.939,-84.556,175.072,26.374,154.543
C04333=1078.528,266.188,-84.584,175.074,26.378,154.544
C04334=1078.533,266.436,-84.614,175.077,26.381,154.544
C04335=1078.539,266.684,-84.641,175.080,26.385,154.545
C04336=1078.545,266.933,-84.671,175.082,26.389,154.545
C04337=1078.551,267.181,-84.699,175.085,26.393,154.546
C04338=1078.556,267.429,-84.727,175.087,26.396,154.546
C04339=1078.562,267.678,-84.756,175.091,26.400,154.547
C04340=1078.568,267.926,-84.784,175.093,26.404,154.547
C04341=1078.574,268.174,-84.813,175.096,26.408,154.548
C04342=1078.579,268.423,-84.842,175.098,26.411,154.548
C04343=1078.585,268.671,-84.871,175.100,26.415,154.549
C04344=1078.591,268.919,-84.899,175.104,26.419,154.550
C04345=1078.597,269.167,-84.928,175.106,26.422,154.550
C04346=1078.603,269.415,-84.957,175.109,26.426,154.551
C04347=1078.608,269.664,-84.986,175.111,26.430,154.551
C04348=1078.614,269.912,-85.014,175.114,26.433,154.552
C04349=1078.620,270.160,-85.043,175.117,26.437,154.552
C04350=1078.626,270.409,-85.072,175.120,26.441,154.553
C04351=1078.632,270.657,-85.101,175.122,26.444,154.553
C04352=1078.637,270.905,-85.129,175.125,26.448,154.554
C04353=1078.643,271.153,-85.158,175.127,26.452,154.554
C04354=1078.650,271.401,-85.187,175.130,26.456,154.555
C04355=1078.655,271.650,-85.216,175.133,26.460,154.555
C04356=1078.660,271.898,-85.245,175.135,26.463,154.556
C04357=1078.667,272.146,-85.274,175.138,26.467,154.556
C04358=1078.672,272.395,-85.303,175.140,26.471,154.557
C04359=1078.678,272.643,-85.332,175.143,26.475,154.557
C04360=1078.684,272.891,-85.361,175.146,26.478,154.558
C04361=1078.689,273.139,-85.390,175.149,26.482,154.558
C04362=1078.695,273.388,-85.419,175.151,26.486,154.559
C04363=1078.701,273.636,-85.448,175.154,26.489,154.560
C04364=1078.707,273.884,-85.477,175.156,26.493,154.560
C04365=1078.713,274.133,-85.506,175.159,26.497,154.561
C04366=1078.718,274.380,-85.536,175.162,26.501,154.561
C04367=1078.724,274.628,-85.565,175.165,26.505,154.562
C04368=1078.730,274.877,-85.594,175.167,26.508,154.562
C04369=1078.736,275.126,-85.623,175.170,26.512,154.563
C04370=1078.742,275.374,-85.652,175.172,26.516,154.563
C04371=1078.748,275.622,-85.681,175.176,26.520,154.564
C04372=1078.757,276.018,-85.728,175.179,26.525,154.565
C04373=1078.766,276.413,-85.775,175.184,26.532,154.566
C04374=1078.775,276.809,-85.822,175.189,26.538,154.566
C04375=1078.784,277.205,-85.868,175.192,26.544,154.567
C04376=1078.790,277.454,-85.897,175.196,26.548,154.568
C04377=1078.796,277.701,-85.927,175.198,26.552,154.568
C04378=1078.802,277.950,-85.956,175.201,26.555,154.569
C04379=1078.808,278.198,-85.986,175.203,26.559,154.570
C04380=1078.813,278.446,-86.015,175.206,26.563,154.570
C04381=1078.819,278.695,-86.044,175.208,26.566,154.571
C04382=1078.825,278.943,-86.074,175.212,26.570,154.571
C04383=1078.831,279.191,-86.103,175.214,26.574,154.572
C04384=1078.837,279.440,-86.133,175.217,26.578,154.572
C04385=1078.842,279.687,-86.161,175.219,26.582,154.573
C04386=1078.848,279.935,-86.192,175.222,26.586,154.573
C04387=1078.854,280.183,-86.221,175.226,26.589,154.574
C04388=1078.860,280.431,-86.251,175.228,26.593,154.574
C04389=1078.865,280.680,-86.280,175.231,26.597,154.575
C04390=1078.872,280.928,-86.309,175.233,26.601,154.575
C04391=1078.878,281.176,-86.340,175.236,26.605,154.576
C04392=1078.883,281.424,-86.369,175.238,26.608,154.577
C04393=1078.889,281.673,-86.399,175.242,26.613,154.577
C04394=1078.895,281.921,-86.428,175.244,26.616,154.578
C04395=1078.901,282.169,-86.458,175.247,26.620,154.578
C04396=1078.906,282.417,-86.488,175.249,26.624,154.579
C04397=1078.912,282.666,-86.517,175.252,26.628,154.579
C04398=1078.917,282.913,-86.548,175.255,26.632,154.580
C04399=1078.924,283.161,-86.577,175.258,26.635,154.580
C04400=1078.930,283.409,-86.607,175.261,26.640,154.581
C04401=1078.935,283.658,-86.637,175.263,26.643,154.582
C04402=1078.941,283.906,-86.666,175.266,26.647,154.582
C04403=1078.946,284.154,-86.697,175.268,26.651,154.583
C04404=1078.953,284.402,-86.726,175.272,26.655,154.583
C04405=1078.958,284.650,-86.756,175.274,26.658,154.584
C04406=1078.964,284.898,-86.786,175.277,26.662,154.584
C04407=1078.970,285.146,-86.816,175.280,26.667,154.585
C04408=1078.975,285.395,-86.846,175.282,26.670,154.586
C04409=1078.981,285.642,-86.876,175.285,26.674,154.586
C04410=1078.987,285.891,-86.905,175.288,26.678,154.587
C04411=1078.993,286.138,-86.936,175.291,26.682,154.587
C04412=1078.999,286.387,-86.965,175.294,26.686,154.588
C04413=1079.004,286.635,-86.996,175.296,26.690,154.588
C04414=1079.010,286.883,-87.025,175.299,26.694,154.589
C04415=1079.016,287.132,-87.056,175.302,26.697,154.589
C04416=1079.023,287.379,-87.086,175.305,26.701,154.590
C04417=1079.028,287.628,-87.115,175.308,26.705,154.591
C04418=1079.034,287.875,-87.146,175.310,26.709,154.591
C04419=1079.040,288.123,-87.176,175.313,26.713,154.592
C04420=1079.046,288.372,-87.206,175.315,26.717,154.592
C04421=1079.051,288.620,-87.236,175.319,26.721,154.593
C04422=1079.057,288.867,-87.266,175.322,26.724,154.593
C04423=1079.063,289.117,-87.296,175.324,26.728,154.594
C04424=1079.073,289.521,-87.345,175.329,26.734,154.595
C04425=1079.082,289.927,-87.396,175.333,26.741,154.596
C04426=1079.093,290.333,-87.445,175.338,26.747,154.597
C04427=1079.101,290.739,-87.494,175.343,26.754,154.598
C04428=1079.107,290.987,-87.524,175.345,26.757,154.598
C04429=1079.113,291.235,-87.555,175.348,26.762,154.599
C04430=1079.119,291.483,-87.586,175.351,26.766,154.599
C04431=1079.125,291.731,-87.616,175.353,26.770,154.600
C04432=1079.131,291.979,-87.646,175.356,26.774,154.601
C04433=1079.137,292.227,-87.677,175.360,26.778,154.601
C04434=1079.143,292.476,-87.707,175.362,26.781,154.602
C04435=1079.148,292.724,-87.738,175.365,26.786,154.602
C04436=1079.154,292.972,-87.768,175.367,26.789,154.603
C04437=1079.160,293.220,-87.798,175.370,26.793,154.603
C04438=1079.165,293.467,-87.829,175.373,26.797,154.604
C04439=1079.172,293.716,-87.859,175.376,26.801,154.605
C04440=1079.178,293.964,-87.890,175.379,26.805,154.605
C04441=1079.183,294.212,-87.921,175.382,26.809,154.606
C04442=1079.188,294.460,-87.951,175.384,26.813,154.606
C04443=1079.195,294.708,-87.982,175.387,26.817,154.607
C04444=1079.201,294.955,-88.013,175.390,26.821,154.608
C04445=1079.207,295.203,-88.043,175.393,26.825,154.608
C04446=1079.213,295.451,-88.073,175.396,26.829,154.609
C04447=1079.218,295.700,-88.105,175.399,26.833,154.609
C04448=1079.224,295.948,-88.135,175.401,26.837,154.610
C04449=1079.230,296.196,-88.165,175.404,26.841,154.610
C04450=1079.236,296.444,-88.196,175.408,26.845,154.611
C04451=1079.242,296.692,-88.228,175.410,26.849,154.612
C04452=1079.248,296.939,-88.258,175.413,26.853,154.612
C04453=1079.253,297.187,-88.289,175.416,26.857,154.613
C04454=1079.259,297.436,-88.320,175.418,26.861,154.613
C04455=1079.265,297.684,-88.350,175.421,26.865,154.614
C04456=1079.271,297.931,-88.381,175.425,26.869,154.615
C04457=1079.277,298.180,-88.413,175.427,26.873,154.615
C04458=1079.283,298.428,-88.443,175.430,26.877,154.616
C04459=1079.288,298.675,-88.475,175.433,26.882,154.617
C04460=1079.294,298.923,-88.505,175.435,26.885,154.617
C04461=1079.299,299.172,-88.536,175.438,26.889,154.618
C04462=1079.306,299.419,-88.567,175.441,26.894,154.618
C04463=1079.311,299.667,-88.598,175.445,26.898,154.619
C04464=1079.317,299.916,-88.629,175.447,26.901,154.620
C04465=1079.322,300.163,-88.661,175.450,26.906,154.620
C04466=1079.327,300.411,-88.692,175.453,26.910,154.621
C04467=1079.334,300.659,-88.723,175.455,26.914,154.621
C04468=1079.339,300.907,-88.754,175.458,26.918,154.622
C04469=1079.345,301.155,-88.785,175.462,26.922,154.623
C04470=1079.350,301.403,-88.816,175.464,26.926,154.623
C04471=1079.357,301.651,-88.847,175.467,26.931,154.624
C04472=1079.362,301.899,-88.878,175.470,26.935,154.625
C04473=1079.368,302.147,-88.910,175.473,26.939,154.625
C04474=1079.374,302.395,-88.941,175.475,26.943,154.626
C04475=1079.379,302.642,-88.972,175.478,26.947,154.626
C04476=1079.385,302.852,-88.999,175.481,26.951,154.627
C04477=1079.390,303.063,-89.025,175.483,26.954,154.627
C04478=1079.395,303.273,-89.052,175.486,26.958,154.628
C04479=1079.399,303.483,-89.079,175.489,26.961,154.629
C04480=1079.404,303.693,-89.105,175.491,26.965,154.629
C04481=1079.409,303.903,-89.132,175.493,26.968,154.630
C04482=1079.415,304.113,-89.158,175.496,26.971,154.630
C04483=1079.419,304.324,-89.185,175.498,26.975,154.631
C04484=1079.425,304.571,-89.216,175.501,26.979,154.631
C04485=1079.431,304.819,-89.248,175.504,26.983,154.632
C04486=1079.436,305.067,-89.279,175.507,26.988,154.633
C04487=1079.443,305.315,-89.310,175.509,26.992,154.633
C04488=1079.448,305.563,-89.342,175.513,26.995,154.634
C04489=1079.455,305.810,-89.373,175.516,27.000,154.634
C04490=1079.460,306.059,-89.404,175.519,27.004,154.635
C04491=1079.466,306.307,-89.436,175.521,27.008,154.636
C04492=1079.472,306.554,-89.467,175.524,27.012,154.636
C04493=1079.478,306.802,-89.499,175.527,27.017,154.637
C04494=1079.483,307.050,-89.531,175.530,27.020,154.637
C04495=1079.489,307.298,-89.563,175.533,27.024,154.638
C04496=1079.495,307.546,-89.593,175.536,27.029,154.639
C04497=1079.501,307.794,-89.625,175.539,27.033,154.639
C04498=1079.507,308.041,-89.657,175.542,27.037,154.640
C04499=1079.513,308.289,-89.688,175.545,27.042,154.641
C04500=1079.519,308.538,-89.720,175.547,27.046,154.641
C04501=1079.525,308.785,-89.752,175.551,27.050,154.642
C04502=1079.531,309.033,-89.784,175.554,27.054,154.643
C04503=1079.537,309.280,-89.815,175.557,27.058,154.643
C04504=1079.543,309.529,-89.847,175.560,27.062,154.644
C04505=1079.549,309.777,-89.879,175.562,27.066,154.644
C04506=1079.555,310.024,-89.910,175.565,27.071,154.645
C04507=1079.561,310.272,-89.942,175.568,27.075,154.646
C04508=1079.567,310.521,-89.974,175.572,27.079,154.646
C04509=1079.572,310.768,-90.006,175.574,27.083,154.647
C04510=1079.579,311.016,-90.037,175.577,27.087,154.648
C04511=1079.585,311.264,-90.069,175.580,27.091,154.648
C04512=1079.590,311.512,-90.101,175.583,27.096,154.649
C04513=1079.596,311.760,-90.133,175.586,27.100,154.650
C04514=1079.603,312.008,-90.166,175.589,27.104,154.650
C04515=1079.609,312.255,-90.197,175.592,27.108,154.651
C04516=1079.615,312.503,-90.229,175.595,27.112,154.652
C04517=1079.621,312.751,-90.261,175.598,27.117,154.652
C04518=1079.627,312.999,-90.293,175.601,27.121,154.653
C04519=1079.632,313.247,-90.325,175.604,27.125,154.653
C04520=1079.639,313.494,-90.357,175.607,27.129,154.654
C04521=1079.645,313.742,-90.389,175.610,27.134,154.655
C04522=1079.651,313.991,-90.421,175.613,27.138,154.655
C04523=1079.657,314.239,-90.453,175.616,27.142,154.656
C04524=1079.663,314.486,-90.485,175.619,27.146,154.657
C04525=1079.669,314.734,-90.517,175.622,27.151,154.657
C04526=1079.675,314.982,-90.549,175.624,27.155,154.658
C04527=1079.681,315.230,-90.582,175.628,27.159,154.659
C04528=1079.686,315.477,-90.614,175.631,27.164,154.659
C04529=1079.692,315.726,-90.646,175.634,27.168,154.660
C04530=1079.698,315.973,-90.679,175.637,27.172,154.661
C04531=1079.703,316.221,-90.711,175.639,27.177,154.662
C04532=1079.708,316.432,-90.739,175.642,27.181,154.662
C04533=1079.714,316.644,-90.766,175.645,27.184,154.663
C04534=1079.718,316.855,-90.794,175.647,27.188,154.663
C04535=1079.723,317.068,-90.822,175.650,27.192,154.664
C04536=1079.728,317.279,-90.849,175.652,27.196,154.664
C04537=1079.733,317.491,-90.877,175.655,27.199,154.665
C04538=1079.738,317.702,-90.905,175.657,27.203,154.666
C04539=1079.743,317.913,-90.933,175.660,27.207,154.666
C04540=1079.749,318.162,-90.965,175.663,27.211,154.667
C04541=1079.755,318.410,-90.998,175.665,27.216,154.668
C04542=1079.760,318.657,-91.030,175.669,27.220,154.668
C04543=1079.766,318.905,-91.063,175.672,27.225,154.669
C04544=1079.772,319.153,-91.095,175.675,27.229,154.670
C04545=1079.778,319.401,-91.128,175.678,27.233,154.670
C04546=1079.784,319.648,-91.161,175.681,27.238,154.671
C04547=1079.790,319.897,-91.193,175.684,27.242,154.672
C04548=1079.795,320.144,-91.226,175.686,27.247,154.673
C04549=1079.802,320.391,-91.258,175.689,27.251,154.673
C04550=1079.807,320.640,-91.291,175.693,27.255,154.674
C04551=1079.813,320.887,-91.324,175.696,27.260,154.675
C04552=1079.819,321.135,-91.357,175.699,27.264,154.675
C04553=1079.825,321.383,-91.390,175.702,27.269,154.676
C04554=1079.831,321.631,-91.422,175.705,27.273,154.677
C04555=1079.837,321.879,-91.455,175.708,27.278,154.677
C04556=1079.842,322.126,-91.488,175.711,27.282,154.678
C04557=1079.848,322.374,-91.520,175.713,27.287,154.679
C04558=1079.855,322.621,-91.553,175.717,27.291,154.680
C04559=1079.860,322.870,-91.586,175.720,27.296,154.680
C04560=1079.866,323.117,-91.618,175.723,27.300,154.681
C04561=1079.872,323.365,-91.652,175.726,27.305,154.682
C04562=1079.878,323.613,-91.685,175.729,27.309,154.682
C04563=1079.884,323.860,-91.717,175.732,27.314,154.683
C04564=1079.890,324.108,-91.751,175.735,27.318,154.684
C04565=1079.896,324.356,-91.783,175.738,27.323,154.685
C04566=1079.902,324.604,-91.817,175.741,27.327,154.685
C04567=1079.908,324.851,-91.849,175.745,27.332,154.686
C04568=1079.914,325.099,-91.883,175.747,27.336,154.687
C04569=1079.920,325.347,-91.916,175.750,27.341,154.687
C04570=1079.926,325.594,-91.948,175.753,27.345,154.688
C04571=1079.932,325.842,-91.982,175.756,27.350,154.689
C04572=1079.938,326.090,-92.014,175.759,27.355,154.690
C04573=1079.944,326.338,-92.048,175.762,27.359,154.690
C04574=1079.950,326.585,-92.080,175.765,27.364,154.691
C04575=1079.956,326.834,-92.114,175.769,27.368,154.692
C04576=1079.962,327.082,-92.147,175.772,27.373,154.693
C04577=1079.968,327.330,-92.180,175.775,27.377,154.693
C04578=1079.974,327.577,-92.213,175.778,27.382,154.694
C04579=1079.980,327.825,-92.246,175.781,27.386,154.695
C04580=1079.986,328.072,-92.280,175.784,27.391,154.696
C04581=1079.992,328.320,-92.313,175.787,27.395,154.696
C04582=1079.998,328.568,-92.346,175.790,27.400,154.697
C04583=1080.004,328.815,-92.379,175.794,27.404,154.698
C04584=1080.011,329.064,-92.412,175.797,27.409,154.698
C04585=1080.017,329.311,-92.446,175.800,27.414,154.699
C04586=1080.023,329.559,-92.479,175.803,27.419,154.700
C04587=1080.028,329.807,-92.512,175.806,27.423,154.701
C04588=1080.039,330.224,-92.569,175.810,27.431,154.702
C04589=1080.050,330.640,-92.625,175.816,27.438,154.703
C04590=1080.059,331.056,-92.681,175.822,27.446,154.704
C04591=1080.070,331.473,-92.737,175.827,27.454,154.706
C04592=1080.076,331.721,-92.771,175.830,27.458,154.706
C04593=1080.082,331.968,-92.805,175.833,27.463,154.707
C04594=1080.087,332.216,-92.838,175.836,27.468,154.708
C04595=1080.094,332.463,-92.872,175.839,27.473,154.709
C04596=1080.100,332.711,-92.905,175.843,27.477,154.709
C04597=1080.106,332.959,-92.939,175.846,27.482,154.710
C04598=1080.112,333.207,-92.973,175.849,27.487,154.711
C04599=1080.117,333.454,-93.007,175.852,27.492,154.712
C04600=1080.123,333.702,-93.040,175.855,27.497,154.713
C04601=1080.129,333.950,-93.074,175.858,27.502,154.713
C04602=1080.136,334.197,-93.108,175.861,27.506,154.714
C04603=1080.142,334.445,-93.141,175.864,27.511,154.715
C04604=1080.147,334.692,-93.175,175.867,27.516,154.716
C04605=1080.153,334.940,-93.209,175.870,27.520,154.717
C04606=1080.159,335.188,-93.243,175.873,27.525,154.717
C04607=1080.165,335.436,-93.277,175.877,27.530,154.718
C04608=1080.171,335.683,-93.311,175.880,27.535,154.719
C04609=1080.177,335.932,-93.345,175.883,27.540,154.720
C04610=1080.183,336.179,-93.379,175.886,27.545,154.721
C04611=1080.189,336.426,-93.413,175.889,27.549,154.721
C04612=1080.196,336.674,-93.447,175.892,27.554,154.722
C04613=1080.202,336.922,-93.480,175.895,27.559,154.723
C04614=1080.208,337.169,-93.514,175.898,27.564,154.724
C04615=1080.214,337.417,-93.549,175.901,27.569,154.725
C04616=1080.220,337.664,-93.583,175.904,27.573,154.725
C04617=1080.226,337.912,-93.617,175.908,27.579,154.726
C04618=1080.232,338.160,-93.651,175.912,27.583,154.727
C04619=1080.238,338.407,-93.684,175.915,27.588,154.728
C04620=1080.243,338.655,-93.719,175.918,27.593,154.729
C04621=1080.249,338.903,-93.754,175.921,27.598,154.729
C04622=1080.255,339.150,-93.788,175.924,27.603,154.730
C04623=1080.261,339.398,-93.822,175.927,27.608,154.731
C04624=1080.268,339.646,-93.856,175.930,27.613,154.732
C04625=1080.274,339.893,-93.890,175.933,27.618,154.733
C04626=1080.279,340.140,-93.924,175.936,27.623,154.734
C04627=1080.286,340.388,-93.959,175.939,27.628,154.734
C04628=1080.291,340.636,-93.993,175.942,27.633,154.735
C04629=1080.297,340.884,-94.028,175.946,27.638,154.736
C04630=1080.304,341.130,-94.062,175.949,27.643,154.737
C04631=1080.309,341.378,-94.096,175.952,27.648,154.738
C04632=1080.316,341.626,-94.131,175.956,27.653,154.739
C04633=1080.322,341.873,-94.165,175.959,27.658,154.739
C04634=1080.328,342.121,-94.200,175.962,27.663,154.740
C04635=1080.333,342.368,-94.234,175.965,27.668,154.741
C04636=1080.340,342.616,-94.268,175.968,27.673,154.742
C04637=1080.346,342.863,-94.303,175.972,27.678,154.743
C04638=1080.352,343.111,-94.338,175.975,27.683,154.744
C04639=1080.358,343.359,-94.372,175.978,27.688,154.744
C04640=1080.368,343.770,-94.429,175.984,27.696,154.746
C04641=1080.378,344.182,-94.487,175.989,27.705,154.747
C04642=1080.389,344.592,-94.545,175.994,27.713,154.749
C04643=1080.398,345.003,-94.602,175.999,27.721,154.750
C04644=1080.405,345.251,-94.637,176.003,27.727,154.751
C04645=1080.410,345.498,-94.672,176.006,27.732,154.752
C04646=1080.416,345.746,-94.706,176.009,27.737,154.753
C04647=1080.422,345.993,-94.742,176.012,27.743,154.754
C04648=1080.428,346.241,-94.776,176.015,27.748,154.755
C04649=1080.434,346.489,-94.812,176.018,27.752,154.755
C04650=1080.440,346.736,-94.846,176.022,27.758,154.756
C04651=1080.447,346.983,-94.881,176.025,27.763,154.757
C04652=1080.452,347.231,-94.916,176.028,27.768,154.758
C04653=1080.459,347.478,-94.951,176.031,27.774,154.759
C04654=1080.464,347.726,-94.985,176.034,27.779,154.760
C04655=1080.471,347.973,-95.021,176.038,27.784,154.761
C04656=1080.477,348.221,-95.056,176.042,27.789,154.762
C04657=1080.483,348.468,-95.090,176.045,27.795,154.763
C04658=1080.489,348.716,-95.126,176.048,27.800,154.764
C04659=1080.495,348.963,-95.161,176.051,27.805,154.765
C04660=1080.501,349.211,-95.196,176.055,27.810,154.765
C04661=1080.507,349.458,-95.231,176.058,27.816,154.766
C04662=1080.513,349.705,-95.266,176.061,27.821,154.767
C04663=1080.519,349.953,-95.301,176.064,27.826,154.768
C04664=1080.525,350.201,-95.337,176.067,27.831,154.769
C04665=1080.531,350.448,-95.372,176.071,27.837,154.770
C04666=1080.537,350.695,-95.407,176.074,27.842,154.771
C04667=1080.544,350.943,-95.443,176.077,27.848,154.772
C04668=1080.549,351.190,-95.477,176.080,27.853,154.773
C04669=1080.555,351.438,-95.513,176.084,27.858,154.774
C04670=1080.562,351.685,-95.548,176.087,27.863,154.775
C04671=1080.568,351.933,-95.583,176.090,27.869,154.776
C04672=1080.574,352.180,-95.619,176.093,27.874,154.777
C04673=1080.580,352.427,-95.654,176.097,27.880,154.777
C04674=1080.586,352.675,-95.690,176.100,27.885,154.778
C04675=1080.592,352.922,-95.725,176.103,27.891,154.779
C04676=1080.599,353.169,-95.760,176.106,27.896,154.780
C04677=1080.605,353.417,-95.796,176.110,27.902,154.781
C04678=1080.611,353.665,-95.832,176.113,27.907,154.782
C04679=1080.616,353.912,-95.867,176.117,27.912,154.783
C04680=1080.623,354.159,-95.902,176.120,27.918,154.784
C04681=1080.629,354.407,-95.938,176.124,27.923,154.785
C04682=1080.635,354.654,-95.974,176.127,27.929,154.786
C04683=1080.640,354.901,-96.009,176.130,27.935,154.787
C04684=1080.646,355.149,-96.045,176.134,27.940,154.788
C04685=1080.653,355.396,-96.080,176.137,27.946,154.789
C04686=1080.659,355.643,-96.116,176.140,27.951,154.790
C04687=1080.666,355.891,-96.152,176.143,27.957,154.791
C04688=1080.671,356.138,-96.187,176.147,27.962,154.792
C04689=1080.677,356.386,-96.223,176.150,27.968,154.793
C04690=1080.684,356.632,-96.259,176.153,27.973,154.794
C04691=1080.690,356.880,-96.295,176.157,27.979,154.795
C04692=1080.700,357.295,-96.355,176.162,27.988,154.797
C04693=1080.710,357.709,-96.415,176.168,27.997,154.798
C04694=1080.721,358.123,-96.474,176.173,28.007,154.800
C04695=1080.731,358.537,-96.535,176.179,28.017,154.802
C04696=1080.737,358.785,-96.571,176.182,28.022,154.803
C04697=1080.743,359.032,-96.607,176.185,28.027,154.804
C04698=1080.749,359.279,-96.643,176.189,28.033,154.805
C04699=1080.755,359.527,-96.679,176.192,28.039,154.806
C04700=1080.762,359.774,-96.715,176.195,28.045,154.807
C04701=1080.768,360.022,-96.751,176.199,28.051,154.808
C04702=1080.774,360.269,-96.787,176.202,28.056,154.809
C04703=1080.780,360.515,-96.823,176.205,28.062,154.810
C04704=1080.786,360.763,-96.859,176.209,28.068,154.811
C04705=1080.792,361.010,-96.896,176.212,28.073,154.812
C04706=1080.798,361.258,-96.931,176.216,28.079,154.813
C04707=1080.805,361.505,-96.968,176.219,28.085,154.814
C04708=1080.811,361.752,-97.004,176.222,28.091,154.815
C04709=1080.817,361.999,-97.040,176.226,28.097,154.816
C04710=1080.823,362.246,-97.076,176.229,28.103,154.817
C04711=1080.830,362.494,-97.113,176.232,28.108,154.818
C04712=1080.836,362.741,-97.149,176.236,28.114,154.819
C04713=1080.842,362.988,-97.185,176.239,28.120,154.820
C04714=1080.848,363.235,-97.222,176.243,28.126,154.821
C04715=1080.854,363.483,-97.259,176.246,28.132,154.822
C04716=1080.860,363.730,-97.295,176.249,28.138,154.823
C04717=1080.866,363.977,-97.331,176.253,28.144,154.824
C04718=1080.873,364.224,-97.367,176.256,28.149,154.825
C04719=1080.879,364.472,-97.404,176.260,28.156,154.827
C04720=1080.885,364.719,-97.440,176.263,28.161,154.828
C04721=1080.892,364.967,-97.477,176.266,28.167,154.829
C04722=1080.898,365.214,-97.514,176.270,28.173,154.830
C04723=1080.904,365.461,-97.550,176.273,28.179,154.831
C04724=1080.911,365.708,-97.587,176.277,28.185,154.832
C04725=1080.916,365.955,-97.624,176.280,28.191,154.833
C04726=1080.922,366.202,-97.660,176.284,28.197,154.834
C04727=1080.928,366.450,-97.697,176.287,28.203,154.835
C04728=1080.934,366.697,-97.734,176.290,28.209,154.836
C04729=1080.941,366.944,-97.770,176.294,28.215,154.837
C04730=1080.946,367.191,-97.807,176.297,28.222,154.839
C04731=1080.953,367.438,-97.844,176.301,28.228,154.840
C04732=1080.959,367.685,-97.880,176.304,28.234,154.841
C04733=1080.966,367.933,-97.918,176.308,28.240,154.842
C04734=1080.972,368.180,-97.955,176.311,28.246,154.843
C04735=1080.977,368.427,-97.992,176.315,28.253,154.844
C04736=1080.984,368.674,-98.028,176.318,28.258,154.845
C04737=1080.990,368.921,-98.065,176.321,28.264,154.846
C04738=1080.996,369.168,-98.102,176.325,28.271,154.848
C04739=1081.002,369.415,-98.139,176.328,28.277,154.849
C04740=1081.009,369.663,-98.176,176.332,28.283,154.850
C04741=1081.015,369.909,-98.213,176.335,28.289,154.851
C04742=1081.021,370.157,-98.250,176.339,28.296,154.852
C04743=1081.027,370.404,-98.287,176.342,28.302,154.853
C04744=1081.033,370.619,-98.319,176.345,28.307,154.854
C04745=1081.039,370.834,-98.352,176.348,28.312,154.855
C04746=1081.044,371.049,-98.384,176.351,28.318,154.856
C04747=1081.049,371.265,-98.416,176.354,28.324,154.857
C04748=1081.055,371.480,-98.449,176.357,28.329,154.858
C04749=1081.060,371.695,-98.481,176.360,28.334,154.859
C04750=1081.065,371.910,-98.514,176.363,28.340,154.860
C04751=1081.072,372.125,-98.546,176.366,28.346,154.862
C04752=1081.077,372.373,-98.583,176.369,28.352,154.863
C04753=1081.084,372.619,-98.620,176.373,28.358,154.864
C04754=1081.089,372.866,-98.658,176.376,28.364,154.865
C04755=1081.097,373.114,-98.695,176.380,28.371,154.866
C04756=1081.103,373.360,-98.733,176.383,28.377,154.867
C04757=1081.109,373.608,-98.770,176.387,28.383,154.869
C04758=1081.115,373.855,-98.807,176.391,28.390,154.870
C04759=1081.121,374.102,-98.844,176.394,28.396,154.871
C04760=1081.128,374.349,-98.882,176.398,28.403,154.872
C04761=1081.134,374.596,-98.920,176.401,28.409,154.873
C04762=1081.140,374.843,-98.957,176.405,28.416,154.875
C04763=1081.146,375.090,-98.994,176.408,28.422,154.876
C04764=1081.153,375.337,-99.032,176.412,28.429,154.877
C04765=1081.159,375.584,-99.070,176.415,28.435,154.878
C04766=1081.165,375.831,-99.108,176.419,28.442,154.880
C04767=1081.171,376.078,-99.146,176.423,28.449,154.881
C04768=1081.177,376.325,-99.183,176.426,28.456,154.882
C04769=1081.183,376.572,-99.220,176.430,28.462,154.883
C04770=1081.190,376.820,-99.258,176.433,28.468,154.885
C04771=1081.196,377.066,-99.296,176.436,28.475,154.886
C04772=1081.202,377.314,-99.334,176.439,28.482,154.887
C04773=1081.208,377.560,-99.372,176.443,28.489,154.888
C04774=1081.215,377.807,-99.409,176.447,28.495,154.890
C04775=1081.221,378.054,-99.447,176.450,28.502,154.891
C04776=1081.227,378.301,-99.485,176.454,28.508,154.892
C04777=1081.234,378.549,-99.523,176.458,28.515,154.893
C04778=1081.240,378.795,-99.561,176.461,28.522,154.895
C04779=1081.247,379.042,-99.599,176.465,28.529,154.896
C04780=1081.253,379.289,-99.637,176.468,28.535,154.897
C04781=1081.260,379.536,-99.675,176.472,28.542,154.899
C04782=1081.266,379.783,-99.712,176.476,28.549,154.900
C04783=1081.272,380.030,-99.751,176.479,28.555,154.901
C04784=1081.278,380.277,-99.788,176.483,28.563,154.903
C04785=1081.285,380.524,-99.827,176.487,28.570,154.904
C04786=1081.291,380.770,-99.865,176.490,28.576,154.905
C04787=1081.297,381.018,-99.903,176.493,28.583,154.906
C04788=1081.304,381.264,-99.940,176.497,28.590,154.908
C04789=1081.311,381.511,-99.979,176.500,28.597,154.909
C04790=1081.317,381.759,-100.017,176.504,28.604,154.910
C04791=1081.323,382.005,-100.055,176.508,28.611,154.912
C04792=1081.330,382.252,-100.094,176.511,28.618,154.913
C04793=1081.336,382.499,-100.131,176.515,28.624,154.914
C04794=1081.343,382.746,-100.170,176.519,28.632,154.916
C04795=1081.348,382.993,-100.209,176.522,28.638,154.917
C04796=1081.355,383.240,-100.247,176.526,28.646,154.919
C04797=1081.360,383.486,-100.285,176.530,28.653,154.920
C04798=1081.367,383.733,-100.324,176.533,28.659,154.921
C04799=1081.374,383.981,-100.362,176.536,28.667,154.923
C04800=1081.379,384.209,-100.398,176.540,28.673,154.924
C04801=1081.385,384.439,-100.434,176.543,28.680,154.925
C04802=1081.391,384.668,-100.470,176.546,28.687,154.926
C04803=1081.397,384.898,-100.505,176.550,28.693,154.928
C04804=1081.403,385.127,-100.541,176.553,28.700,154.929
C04805=1081.408,385.357,-100.577,176.556,28.706,154.930
C04806=1081.415,385.586,-100.613,176.560,28.713,154.932
C04807=1081.420,385.816,-100.649,176.563,28.720,154.933
C04808=1081.427,386.063,-100.688,176.567,28.727,154.934
C04809=1081.434,386.309,-100.727,176.571,28.735,154.936
C04810=1081.439,386.556,-100.765,176.575,28.742,154.937
C04811=1081.446,386.803,-100.803,176.578,28.749,154.939
C04812=1081.452,387.050,-100.843,176.582,28.756,154.940
C04813=1081.459,387.296,-100.881,176.586,28.764,154.942
C04814=1081.465,387.543,-100.920,176.590,28.771,154.943
C04815=1081.472,387.790,-100.959,176.593,28.778,154.944
C04816=1081.478,388.037,-100.998,176.596,28.786,154.946
C04817=1081.485,388.283,-101.037,176.600,28.793,154.947
C04818=1081.491,388.531,-101.075,176.604,28.800,154.949
C04819=1081.497,388.778,-101.114,176.608,28.808,154.950
C04820=1081.504,389.025,-101.153,176.611,28.815,154.952
C04821=1081.511,389.271,-101.192,176.615,28.822,154.953
C04822=1081.517,389.517,-101.231,176.619,28.830,154.955
C04823=1081.523,389.764,-101.271,176.623,28.837,154.956
C04824=1081.530,390.011,-101.310,176.627,28.845,154.958
C04825=1081.537,390.258,-101.348,176.631,28.852,154.959
C04826=1081.543,390.505,-101.388,176.633,28.860,154.960
C04827=1081.550,390.752,-101.427,176.637,28.867,154.962
C04828=1081.557,390.998,-101.466,176.641,28.875,154.963
C04829=1081.563,391.246,-101.505,176.645,28.883,154.965
C04830=1081.570,391.492,-101.545,176.649,28.890,154.966
C04831=1081.576,391.739,-101.584,176.653,28.898,154.968
C04832=1081.582,391.985,-101.622,176.657,28.905,154.969
C04833=1081.588,392.232,-101.662,176.660,28.913,154.971
C04834=1081.595,392.478,-101.701,176.664,28.921,154.973
C04835=1081.601,392.725,-101.741,176.667,28.928,154.974
C04836=1081.608,392.972,-101.780,176.671,28.936,154.976
C04837=1081.615,393.219,-101.820,176.675,28.944,154.977
C04838=1081.621,393.466,-101.859,176.679,28.952,154.979
C04839=1081.628,393.712,-101.899,176.683,28.960,154.980
C04840=1081.634,393.959,-101.938,176.686,28.967,154.982
C04841=1081.641,394.205,-101.978,176.690,28.975,154.983
C04842=1081.647,394.453,-102.017,176.694,28.983,154.985
C04843=1081.654,394.699,-102.057,176.697,28.991,154.987
C04844=1081.660,394.946,-102.096,176.701,28.999,154.988
C04845=1081.667,395.192,-102.136,176.705,29.007,154.990
C04846=1081.673,395.440,-102.176,176.709,29.015,154.991
C04847=1081.680,395.686,-102.215,176.713,29.023,154.993
C04848=1081.686,395.932,-102.255,176.717,29.031,154.995
C04849=1081.692,396.179,-102.295,176.721,29.039,154.996
C04850=1081.699,396.426,-102.335,176.725,29.047,154.998
C04851=1081.706,396.672,-102.375,176.728,29.055,154.999
C04852=1081.712,396.919,-102.414,176.731,29.063,155.001
C04853=1081.718,397.166,-102.454,176.735,29.071,155.003
C04854=1081.725,397.413,-102.495,176.739,29.079,155.004
C04855=1081.732,397.660,-102.535,176.743,29.087,155.006
C04856=1081.740,397.980,-102.586,176.748,29.098,155.008
C04857=1081.749,398.300,-102.638,176.753,29.108,155.010
C04858=1081.758,398.620,-102.690,176.759,29.119,155.012
C04859=1081.766,398.940,-102.742,176.763,29.129,155.015
C04860=1081.772,399.187,-102.782,176.767,29.138,155.016
C04861=1081.779,399.433,-102.822,176.771,29.146,155.018
C04862=1081.785,399.680,-102.862,176.775,29.155,155.020
C04863=1081.791,399.926,-102.902,176.779,29.163,155.021
C04864=1081.798,400.174,-102.943,176.782,29.171,155.023
C04865=1081.805,400.420,-102.983,176.786,29.180,155.025
C04866=1081.811,400.667,-103.023,176.790,29.188,155.026
C04867=1081.818,400.913,-103.063,176.794,29.196,155.028
C04868=1081.825,401.160,-103.105,176.798,29.205,155.030
C04869=1081.831,401.406,-103.145,176.802,29.213,155.032
C04870=1081.838,401.653,-103.185,176.806,29.222,155.034
C04871=1081.844,401.899,-103.225,176.810,29.230,155.035
C04872=1081.851,402.146,-103.265,176.814,29.239,155.037
C04873=1081.858,402.392,-103.306,176.818,29.248,155.039
C04874=1081.864,402.639,-103.346,176.822,29.256,155.041
C04875=1081.871,402.886,-103.387,176.826,29.264,155.042
C04876=1081.877,403.133,-103.427,176.830,29.273,155.044
C04877=1081.885,403.379,-103.468,176.834,29.282,155.046
C04878=1081.891,403.626,-103.509,176.837,29.290,155.048
C04879=1081.897,403.872,-103.549,176.841,29.299,155.049
C04880=1081.908,404.272,-103.615,176.848,29.314,155.052
C04881=1081.919,404.671,-103.681,176.854,29.328,155.055
C04882=1081.929,405.071,-103.747,176.861,29.342,155.058
C04883=1081.941,405.470,-103.813,176.868,29.356,155.061
C04884=1081.947,405.717,-103.855,176.872,29.365,155.063
C04885=1081.954,405.963,-103.895,176.875,29.374,155.065
C04886=1081.961,406.210,-103.936,176.879,29.383,155.067
C04887=1081.967,406.456,-103.978,176.883,29.392,155.069
C04888=1081.974,406.703,-104.018,176.887,29.401,155.071
C04889=1081.980,406.949,-104.059,176.892,29.410,155.072
C04890=1081.987,407.196,-104.101,176.896,29.419,155.074
C04891=1081.993,407.443,-104.141,176.899,29.428,155.076
C04892=1082.001,407.689,-104.183,176.903,29.437,155.078
C04893=1082.007,407.935,-104.224,176.908,29.446,155.080
C04894=1082.014,408.182,-104.265,176.912,29.456,155.082
C04895=1082.020,408.428,-104.307,176.916,29.465,155.084
C04896=1082.027,408.675,-104.348,176.920,29.474,155.086
C04897=1082.034,408.922,-104.390,176.925,29.484,155.088
C04898=1082.040,409.168,-104.431,176.928,29.493,155.090
C04899=1082.047,409.415,-104.472,176.932,29.502,155.092
C04900=1082.054,409.660,-104.513,176.936,29.511,155.094
C04901=1082.060,409.907,-104.555,176.941,29.521,155.096
C04902=1082.067,410.154,-104.596,176.945,29.530,155.098
C04903=1082.073,410.400,-104.638,176.949,29.539,155.100
C04904=1082.081,410.647,-104.679,176.953,29.549,155.102
C04905=1082.087,410.894,-104.721,176.957,29.559,155.104
C04906=1082.094,411.140,-104.762,176.961,29.568,155.106
C04907=1082.100,411.386,-104.804,176.966,29.578,155.108
C04908=1082.107,411.624,-104.844,176.970,29.587,155.109
C04909=1082.114,411.861,-104.884,176.974,29.596,155.111
C04910=1082.120,412.099,-104.924,176.978,29.605,155.113
C04911=1082.127,412.336,-104.964,176.981,29.614,155.115
C04912=1082.133,412.573,-105.004,176.985,29.623,155.117
C04913=1082.140,412.811,-105.045,176.990,29.633,155.119
C04914=1082.147,413.049,-105.085,176.994,29.642,155.121
C04915=1082.153,413.286,-105.125,176.998,29.652,155.123
C04916=1082.160,413.532,-105.167,177.002,29.661,155.125
C04917=1082.167,413.779,-105.208,177.007,29.671,155.127
C04918=1082.174,414.025,-105.251,177.011,29.681,155.129
C04919=1082.180,414.272,-105.293,177.015,29.691,155.132
C04920=1082.188,414.518,-105.335,177.019,29.700,155.134
C04921=1082.194,414.765,-105.377,177.024,29.710,155.136
C04922=1082.201,415.011,-105.419,177.028,29.720,155.138
C04923=1082.208,415.257,-105.460,177.033,29.731,155.140
C04924=1082.215,415.503,-105.502,177.037,29.740,155.142
C04925=1082.222,415.749,-105.545,177.041,29.750,155.144
C04926=1082.228,415.996,-105.587,177.045,29.760,155.146
C04927=1082.236,416.242,-105.629,177.050,29.771,155.149
C04928=1082.243,416.489,-105.671,177.054,29.781,155.151
C04929=1082.250,416.735,-105.714,177.059,29.791,155.153
C04930=1082.256,416.982,-105.756,177.063,29.801,155.155
C04931=1082.263,417.228,-105.798,177.067,29.811,155.157
C04932=1082.270,417.474,-105.841,177.071,29.821,155.159
C04933=1082.277,417.721,-105.883,177.076,29.832,155.162
C04934=1082.283,417.966,-105.925,177.080,29.842,155.164
C04935=1082.290,418.213,-105.968,177.085,29.852,155.166
C04936=1082.297,418.459,-106.011,177.089,29.862,155.168
C04937=1082.304,418.705,-106.053,177.093,29.873,155.171
C04938=1082.310,418.951,-106.096,177.098,29.883,155.173
C04939=1082.317,419.198,-106.138,177.102,29.894,155.175
C04940=1082.324,419.444,-106.181,177.107,29.905,155.177
C04941=1082.332,419.691,-106.224,177.111,29.915,155.180
C04942=1082.339,419.937,-106.267,177.116,29.925,155.182
C04943=1082.346,420.183,-106.309,177.121,29.936,155.184
C04944=1082.352,420.429,-106.352,177.124,29.946,155.186
C04945=1082.359,420.675,-106.394,177.129,29.957,155.189
C04946=1082.366,420.921,-106.438,177.134,29.968,155.191
C04947=1082.373,421.167,-106.480,177.138,29.979,155.193
C04948=1082.380,421.414,-106.523,177.143,29.989,155.196
C04949=1082.388,421.661,-106.566,177.148,30.000,155.198
C04950=1082.395,421.906,-106.609,177.152,30.011,155.200
C04951=1082.402,422.153,-106.652,177.156,30.022,155.203
C04952=1082.409,422.398,-106.695,177.161,30.033,155.205
C04953=1082.416,422.645,-106.737,177.166,30.044,155.208
C04954=1082.422,422.891,-106.781,177.170,30.054,155.210
C04955=1082.430,423.138,-106.824,177.175,30.065,155.212
C04956=1082.437,423.383,-106.867,177.180,30.077,155.215
C04957=1082.443,423.629,-106.911,177.184,30.088,155.217
C04958=1082.450,423.875,-106.954,177.188,30.099,155.220
C04959=1082.457,424.121,-106.997,177.193,30.110,155.222
C04960=1082.465,424.368,-107.041,177.198,30.121,155.225
C04961=1082.471,424.614,-107.084,177.203,30.132,155.227
C04962=1082.478,424.860,-107.127,177.207,30.143,155.229
C04963=1082.485,425.105,-107.170,177.212,30.155,155.232
C04964=1082.493,425.351,-107.213,177.217,30.166,155.234
C04965=1082.499,425.597,-107.257,177.221,30.177,155.237
C04966=1082.506,425.843,-107.301,177.226,30.189,155.239
C04967=1082.513,426.088,-107.344,177.231,30.200,155.242
C04968=1082.521,426.333,-107.388,177.235,30.211,155.244
C04969=1082.528,426.579,-107.431,177.240,30.223,155.247
C04970=1082.534,426.825,-107.475,177.245,30.234,155.249
C04971=1082.542,427.071,-107.519,177.250,30.246,155.252
C04972=1082.549,427.317,-107.562,177.255,30.258,155.255
C04973=1082.556,427.563,-107.606,177.259,30.269,155.257
C04974=1082.564,427.809,-107.650,177.264,30.281,155.260
C04975=1082.571,428.054,-107.693,177.269,30.293,155.262
C04976=1082.578,428.301,-107.737,177.274,30.304,155.265
C04977=1082.585,428.547,-107.781,177.279,30.316,155.267
C04978=1082.592,428.793,-107.825,177.284,30.328,155.270
C04979=1082.600,429.039,-107.869,177.288,30.340,155.273
C04980=1082.606,429.284,-107.913,177.293,30.352,155.275
C04981=1082.613,429.531,-107.958,177.297,30.363,155.278
C04982=1082.621,429.776,-108.001,177.302,30.375,155.281
C04983=1082.628,430.023,-108.045,177.307,30.387,155.283
C04984=1082.635,430.268,-108.089,177.312,30.399,155.286
C04985=1082.642,430.515,-108.133,177.317,30.412,155.289
C04986=1082.649,430.761,-108.178,177.322,30.424,155.292
C04987=1082.657,431.006,-108.222,177.327,30.436,155.294
C04988=1082.664,431.252,-108.266,177.333,30.449,155.297
C04989=1082.671,431.498,-108.311,177.338,30.461,155.300
C04990=1082.679,431.743,-108.355,177.343,30.473,155.303
C04991=1082.686,431.990,-108.400,177.347,30.485,155.305
C04992=1082.692,432.235,-108.444,177.352,30.498,155.308
C04993=1082.700,432.481,-108.488,177.357,30.510,155.311
C04994=1082.708,432.727,-108.533,177.362,30.523,155.314
C04995=1082.714,432.973,-108.577,177.367,30.535,155.316
C04996=1082.722,433.219,-108.622,177.372,30.548,155.319
C04997=1082.728,433.465,-108.667,177.377,30.560,155.322
C04998=1082.736,433.711,-108.712,177.382,30.573,155.325
C04999=1082.743,433.957,-108.757,177.388,30.586,155.328
C05000=1082.750,434.202,-108.801,177.393,30.599,155.331
C05001=1082.758,434.448,-108.846,177.398,30.611,155.334
C05002=1082.765,434.694,-108.890,177.403,30.624,155.336
C05003=1082.772,434.940,-108.935,177.408,30.637,155.339
C05004=1082.779,435.185,-108.981,177.413,30.650,155.342
C05005=1082.787,435.431,-109.026,177.418,30.663,155.345
C05006=1082.794,435.677,-109.071,177.423,30.676,155.348
C05007=1082.801,435.923,-109.115,177.428,30.689,155.351
C05008=1082.809,436.168,-109.161,177.433,30.702,155.354
C05009=1082.816,436.414,-109.206,177.439,30.715,155.357
C05010=1082.823,436.660,-109.251,177.444,30.728,155.360
C05011=1082.831,436.905,-109.296,177.449,30.741,155.363
C05012=1082.838,437.151,-109.341,177.455,30.755,155.366
C05013=1082.846,437.397,-109.387,177.460,30.768,155.369
C05014=1082.853,437.643,-109.432,177.465,30.781,155.372
C05015=1082.861,437.888,-109.477,177.470,30.794,155.375
C05016=1082.868,438.134,-109.522,177.476,30.808,155.378
C05017=1082.876,438.380,-109.568,177.481,30.821,155.381
C05018=1082.883,438.625,-109.614,177.486,30.834,155.384
C05019=1082.891,438.871,-109.659,177.492,30.848,155.388
C05020=1082.900,439.185,-109.717,177.499,30.866,155.391
C05021=1082.910,439.499,-109.775,177.505,30.883,155.396
C05022=1082.919,439.812,-109.833,177.512,30.900,155.399
C05023=1082.929,440.126,-109.892,177.520,30.919,155.404
C05024=1082.937,440.372,-109.938,177.525,30.932,155.407
C05025=1082.944,440.617,-109.983,177.530,30.946,155.410
C05026=1082.951,440.863,-110.030,177.536,30.960,155.413
C05027=1082.959,441.109,-110.075,177.541,30.974,155.416
C05028=1082.966,441.354,-110.121,177.547,30.988,155.420
C05029=1082.974,441.599,-110.166,177.552,31.002,155.423
C05030=1082.981,441.846,-110.213,177.558,31.016,155.426
C05031=1082.989,442.091,-110.259,177.563,31.031,155.429
C05032=1082.997,442.337,-110.304,177.569,31.045,155.433
C05033=1083.004,442.582,-110.351,177.574,31.059,155.436
C05034=1083.012,442.827,-110.397,177.580,31.074,155.439
C05035=1083.018,443.073,-110.443,177.585,31.088,155.443
C05036=1083.027,443.318,-110.490,177.591,31.102,155.446
C05037=1083.035,443.564,-110.536,177.596,31.117,155.450
C05038=1083.042,443.809,-110.583,177.602,31.132,155.453
C05039=1083.050,444.054,-110.628,177.609,31.146,155.456
C05040=1083.057,444.300,-110.676,177.614,31.161,155.460
C05041=1083.065,444.546,-110.721,177.620,31.176,155.463
C05042=1083.072,444.791,-110.768,177.626,31.190,155.467
C05043=1083.080,445.037,-110.814,177.631,31.205,155.470
C05044=1083.088,445.282,-110.861,177.637,31.220,155.474
C05045=1083.096,445.527,-110.907,177.642,31.235,155.477
C05046=1083.103,445.773,-110.955,177.648,31.250,155.480
C05047=1083.110,446.018,-111.001,177.653,31.265,155.484
C05048=1083.118,446.263,-111.047,177.659,31.280,155.488
C05049=1083.126,446.509,-111.095,177.663,31.295,155.491
C05050=1083.134,446.754,-111.141,177.668,31.310,155.495
C05051=1083.142,447.000,-111.188,177.672,31.325,155.498
C05052=1083.149,447.245,-111.235,177.676,31.339,155.502
C05053=1083.158,447.490,-111.282,177.679,31.354,155.505
C05054=1083.165,447.736,-111.329,177.684,31.369,155.509
C05055=1083.173,447.981,-111.376,177.687,31.384,155.513
C05056=1083.180,448.226,-111.423,177.690,31.399,155.516
C05057=1083.188,448.472,-111.470,177.693,31.414,155.520
C05058=1083.195,448.717,-111.517,177.696,31.428,155.524
C05059=1083.204,448.963,-111.564,177.699,31.443,155.527
C05060=1083.212,449.207,-111.611,177.701,31.458,155.531
C05061=1083.219,449.452,-111.658,177.704,31.472,155.534
C05062=1083.230,449.697,-111.704,177.706,31.486,155.538
C05063=1083.243,449.944,-111.748,177.708,31.499,155.541
C05064=1082.873,449.937,-111.961,177.678,31.675,155.588
C05065=1082.860,449.691,-111.917,177.675,31.662,155.585
C05066=1082.850,449.445,-111.871,177.673,31.649,155.582
C05067=1082.841,449.200,-111.824,177.670,31.634,155.578
C05068=1082.833,448.956,-111.777,177.668,31.620,155.574
C05069=1082.825,448.710,-111.729,177.665,31.605,155.571
C05070=1082.817,448.466,-111.683,177.662,31.590,155.567
C05071=1082.809,448.220,-111.635,177.659,31.575,155.563
C05072=1082.802,447.975,-111.589,177.655,31.560,155.560
C05073=1082.793,447.729,-111.542,177.652,31.545,155.556
C05074=1082.786,447.484,-111.495,177.648,31.531,155.553
C05075=1082.778,447.238,-111.448,177.643,31.516,155.549
C05076=1082.770,446.993,-111.401,177.639,31.501,155.545
C05077=1082.763,446.748,-111.354,177.635,31.486,155.542
C05078=1082.755,446.502,-111.307,177.631,31.471,155.538
C05079=1082.747,446.257,-111.260,177.625,31.456,155.534
C05080=1082.740,446.012,-111.213,177.620,31.441,155.531
C05081=1082.732,445.766,-111.166,177.615,31.426,155.527
C05082=1082.724,445.521,-111.119,177.610,31.411,155.524
C05083=1082.716,445.275,-111.072,177.603,31.396,155.520
C05084=1082.708,445.030,-111.026,177.597,31.381,155.517
C05085=1082.701,444.785,-110.980,177.592,31.366,155.513
C05086=1082.693,444.539,-110.933,177.586,31.351,155.510
C05087=1082.686,444.293,-110.887,177.581,31.337,155.507
C05088=1082.678,444.049,-110.840,177.574,31.322,155.503
C05089=1082.670,443.803,-110.793,177.568,31.307,155.500
C05090=1082.662,443.557,-110.747,177.563,31.293,155.496
C05091=1082.655,443.312,-110.700,177.557,31.278,155.493
C05092=1082.647,443.066,-110.654,177.552,31.264,155.490
C05093=1082.639,442.821,-110.609,177.546,31.249,155.486
C05094=1082.632,442.576,-110.562,177.540,31.235,155.483
C05095=1082.625,442.330,-110.516,177.534,31.220,155.480
C05096=1082.617,442.085,-110.469,177.529,31.206,155.476
C05097=1082.609,441.839,-110.423,177.523,31.192,155.473
C05098=1082.601,441.593,-110.377,177.518,31.178,155.470
C05099=1082.595,441.348,-110.331,177.512,31.164,155.466
C05100=1082.587,441.102,-110.286,177.507,31.150,155.463
C05101=1082.579,440.857,-110.240,177.500,31.136,155.460
C05102=1082.572,440.611,-110.194,177.495,31.122,155.457
C05103=1082.564,440.365,-110.148,177.489,31.108,155.453
C05104=1082.556,440.120,-110.101,177.484,31.094,155.450
C05105=1082.548,439.822,-110.046,177.477,31.077,155.446
C05106=1082.538,439.523,-109.991,177.470,31.060,155.443
C05107=1082.529,439.224,-109.935,177.464,31.044,155.439
C05108=1082.520,438.926,-109.880,177.458,31.027,155.435
C05109=1082.512,438.680,-109.834,177.451,31.013,155.432
C05110=1082.505,438.435,-109.789,177.446,31.000,155.429
C05111=1082.497,438.189,-109.744,177.441,30.987,155.426
C05112=1082.490,437.943,-109.698,177.435,30.973,155.423
C05113=1082.482,437.698,-109.652,177.430,30.960,155.420
C05114=1082.475,437.452,-109.607,177.425,30.946,155.416
C05115=1082.467,437.207,-109.562,177.420,30.933,155.413
C05116=1082.460,436.960,-109.517,177.414,30.920,155.410
C05117=1082.452,436.715,-109.471,177.409,30.907,155.407
C05118=1082.445,436.469,-109.426,177.404,30.893,155.404
C05119=1082.437,436.224,-109.381,177.398,30.880,155.401
C05120=1082.430,435.978,-109.336,177.393,30.867,155.398
C05121=1082.423,435.732,-109.291,177.388,30.854,155.396
C05122=1082.415,435.487,-109.246,177.383,30.841,155.392
C05123=1082.408,435.241,-109.201,177.378,30.828,155.390
C05124=1082.401,434.995,-109.156,177.372,30.815,155.387
C05125=1082.394,434.749,-109.111,177.367,30.803,155.384
C05126=1082.386,434.504,-109.065,177.362,30.790,155.381
C05127=1082.379,434.258,-109.021,177.357,30.777,155.378
C05128=1082.372,434.012,-108.976,177.352,30.764,155.375
C05129=1082.365,433.766,-108.931,177.347,30.751,155.372
C05130=1082.357,433.521,-108.887,177.341,30.738,155.369
C05131=1082.350,433.275,-108.842,177.336,30.726,155.366
C05132=1082.343,433.029,-108.797,177.331,30.713,155.364
C05133=1082.336,432.783,-108.752,177.326,30.701,155.361
C05134=1082.328,432.537,-108.707,177.321,30.688,155.358
C05135=1082.322,432.292,-108.663,177.316,30.676,155.355
C05136=1082.314,432.045,-108.619,177.311,30.664,155.352
C05137=1082.306,431.799,-108.574,177.306,30.651,155.350
C05138=1082.299,431.553,-108.529,177.301,30.639,155.347
C05139=1082.292,431.308,-108.485,177.296,30.627,155.344
C05140=1082.285,431.062,-108.441,177.291,30.614,155.341
C05141=1082.278,430.816,-108.397,177.286,30.602,155.339
C05142=1082.270,430.570,-108.352,177.281,30.590,155.336
C05143=1082.263,430.324,-108.308,177.276,30.578,155.333
C05144=1082.256,430.078,-108.263,177.271,30.566,155.330
C05145=1082.248,429.832,-108.220,177.266,30.554,155.328
C05146=1082.242,429.587,-108.175,177.261,30.542,155.325
C05147=1082.234,429.340,-108.132,177.256,30.530,155.322
C05148=1082.227,429.095,-108.087,177.251,30.518,155.320
C05149=1082.220,428.848,-108.043,177.246,30.506,155.317
C05150=1082.213,428.603,-108.000,177.241,30.494,155.314
C05151=1082.206,428.357,-107.955,177.236,30.482,155.312
C05152=1082.198,428.111,-107.911,177.231,30.470,155.309
C05153=1082.191,427.864,-107.867,177.226,30.459,155.307
C05154=1082.184,427.619,-107.823,177.221,30.447,155.304
C05155=1082.177,427.373,-107.779,177.216,30.435,155.301
C05156=1082.170,427.127,-107.736,177.211,30.424,155.299
C05157=1082.163,426.881,-107.692,177.206,30.412,155.296
C05158=1082.156,426.635,-107.648,177.202,30.401,155.294
C05159=1082.148,426.389,-107.605,177.197,30.389,155.291
C05160=1082.141,426.143,-107.561,177.192,30.378,155.289
C05161=1082.134,425.897,-107.518,177.187,30.366,155.286
C05162=1082.126,425.650,-107.474,177.182,30.355,155.284
C05163=1082.120,425.403,-107.430,177.178,30.343,155.281
C05164=1082.113,425.156,-107.386,177.174,30.332,155.279
C05165=1082.105,424.911,-107.343,177.169,30.321,155.276
C05166=1082.098,424.665,-107.300,177.164,30.310,155.274
C05167=1082.092,424.418,-107.256,177.159,30.298,155.271
C05168=1082.084,424.172,-107.213,177.154,30.287,155.269
C05169=1082.077,423.926,-107.170,177.150,30.276,155.266
C05170=1082.070,423.681,-107.126,177.145,30.265,155.264
C05171=1082.063,423.433,-107.083,177.140,30.254,155.261
C05172=1082.056,423.188,-107.040,177.135,30.243,155.259
C05173=1082.049,422.942,-106.996,177.131,30.232,155.257
C05174=1082.043,422.695,-106.953,177.126,30.221,155.254
C05175=1082.036,422.450,-106.910,177.121,30.210,155.252
C05176=1082.028,422.203,-106.867,177.117,30.199,155.249
C05177=1082.021,421.957,-106.824,177.112,30.188,155.247
C05178=1082.014,421.711,-106.781,177.108,30.177,155.245
C05179=1082.007,421.465,-106.738,177.103,30.166,155.242
C05180=1082.000,421.219,-106.696,177.099,30.155,155.240
C05181=1081.993,420.972,-106.652,177.094,30.145,155.238
C05182=1081.986,420.726,-106.609,177.089,30.134,155.235
C05183=1081.980,420.480,-106.566,177.085,30.124,155.233
C05184=1081.973,420.233,-106.524,177.080,30.113,155.231
C05185=1081.966,419.988,-106.480,177.076,30.103,155.228
C05186=1081.959,419.741,-106.438,177.071,30.092,155.226
C05187=1081.952,419.495,-106.395,177.066,30.081,155.224
C05188=1081.945,419.249,-106.353,177.062,30.071,155.222
C05189=1081.937,419.003,-106.311,177.057,30.060,155.219
C05190=1081.930,418.756,-106.267,177.054,30.050,155.217
C05191=1081.923,418.510,-106.225,177.049,30.039,155.215
C05192=1081.916,418.264,-106.182,177.044,30.029,155.212
C05193=1081.909,418.018,-106.140,177.040,30.019,155.210
C05194=1081.902,417.771,-106.097,177.035,30.008,155.208
C05195=1081.895,417.525,-106.055,177.031,29.998,155.206
C05196=1081.888,417.279,-106.012,177.026,29.988,155.204
C05197=1081.882,417.033,-105.970,177.022,29.977,155.201
C05198=1081.876,416.786,-105.928,177.017,29.967,155.199
C05199=1081.869,416.540,-105.885,177.013,29.957,155.197
C05200=1081.862,416.294,-105.843,177.008,29.947,155.195
C05201=1081.855,416.047,-105.800,177.005,29.937,155.193
C05202=1081.848,415.801,-105.758,177.000,29.927,155.191
C05203=1081.841,415.554,-105.717,176.996,29.917,155.188
C05204=1081.834,415.308,-105.674,176.991,29.906,155.186
C05205=1081.827,415.062,-105.632,176.987,29.897,155.184
C05206=1081.820,414.815,-105.590,176.982,29.887,155.182
C05207=1081.813,414.569,-105.548,176.978,29.877,155.180
C05208=1081.806,414.323,-105.505,176.973,29.867,155.178
C05209=1081.800,414.077,-105.464,176.969,29.857,155.176
C05210=1081.793,413.831,-105.422,176.965,29.847,155.174
C05211=1081.786,413.584,-105.380,176.961,29.838,155.172
C05212=1081.779,413.338,-105.338,176.957,29.828,155.169
C05213=1081.773,413.099,-105.298,176.953,29.818,155.167
C05214=1081.765,412.861,-105.257,176.948,29.809,155.166
C05215=1081.759,412.623,-105.217,176.944,29.800,155.163
C05216=1081.753,412.385,-105.176,176.940,29.791,155.162
C05217=1081.746,412.147,-105.136,176.936,29.781,155.159
C05218=1081.739,411.909,-105.096,176.932,29.772,155.158
C05219=1081.732,411.670,-105.056,176.927,29.763,155.156
C05220=1081.726,411.432,-105.015,176.923,29.753,155.154
C05221=1081.719,411.186,-104.974,176.919,29.744,155.152
C05222=1081.713,410.940,-104.932,176.915,29.735,155.150
C05223=1081.706,410.693,-104.891,176.910,29.725,155.148
C05224=1081.699,410.446,-104.849,176.907,29.715,155.146
C05225=1081.692,410.200,-104.808,176.903,29.706,155.144
C05226=1081.686,409.953,-104.766,176.898,29.696,155.142
C05227=1081.679,409.707,-104.724,176.894,29.687,155.140
C05228=1081.672,409.461,-104.683,176.890,29.678,155.138
C05229=1081.666,409.214,-104.641,176.886,29.669,155.136
C05230=1081.658,408.968,-104.600,176.881,29.659,155.134
C05231=1081.652,408.722,-104.558,176.877,29.650,155.132
C05232=1081.645,408.475,-104.517,176.873,29.641,155.130
C05233=1081.639,408.228,-104.477,176.869,29.632,155.128
C05234=1081.632,407.982,-104.435,176.865,29.622,155.126
C05235=1081.625,407.736,-104.394,176.861,29.613,155.124
C05236=1081.619,407.489,-104.353,176.857,29.604,155.122
C05237=1081.612,407.242,-104.311,176.853,29.595,155.120
C05238=1081.606,406.996,-104.270,176.849,29.586,155.118
C05239=1081.599,406.749,-104.229,176.844,29.577,155.116
C05240=1081.592,406.503,-104.188,176.840,29.567,155.115
C05241=1081.585,406.256,-104.147,176.836,29.559,155.113
C05242=1081.579,406.010,-104.106,176.832,29.550,155.111
C05243=1081.572,405.763,-104.065,176.828,29.541,155.109
C05244=1081.565,405.517,-104.024,176.824,29.532,155.107
C05245=1081.559,405.270,-103.983,176.820,29.523,155.105
C05246=1081.552,405.024,-103.942,176.816,29.514,155.103
C05247=1081.545,404.777,-103.901,176.812,29.505,155.102
C05248=1081.539,404.530,-103.861,176.808,29.496,155.100
C05249=1081.532,404.283,-103.819,176.804,29.488,155.098
C05250=1081.526,404.037,-103.779,176.800,29.479,155.096
C05251=1081.519,403.791,-103.738,176.796,29.470,155.094
C05252=1081.512,403.544,-103.698,176.792,29.461,155.092
C05253=1081.506,403.297,-103.658,176.787,29.452,155.091
C05254=1081.498,403.051,-103.616,176.784,29.444,155.089
C05255=1081.492,402.804,-103.576,176.780,29.436,155.087
C05256=1081.485,402.558,-103.535,176.776,29.427,155.085
C05257=1081.478,402.311,-103.495,176.772,29.418,155.084
C05258=1081.472,402.065,-103.455,176.768,29.410,155.082
C05259=1081.466,401.818,-103.414,176.764,29.401,155.080
C05260=1081.459,401.571,-103.373,176.760,29.393,155.078
C05261=1081.453,401.325,-103.333,176.756,29.384,155.077
C05262=1081.446,401.078,-103.292,176.752,29.376,155.075
C05263=1081.439,400.831,-103.252,176.748,29.367,155.073
C05264=1081.433,400.584,-103.212,176.744,29.359,155.071
C05265=1081.426,400.338,-103.172,176.740,29.351,155.070
C05266=1081.420,400.091,-103.131,176.737,29.342,155.068
C05267=1081.413,399.845,-103.090,176.733,29.334,155.066
C05268=1081.406,399.598,-103.050,176.729,29.325,155.064
C05269=1081.400,399.361,-103.012,176.725,29.317,155.063
C05270=1081.394,399.124,-102.974,176.721,29.309,155.061
C05271=1081.387,398.887,-102.935,176.718,29.301,155.060
C05272=1081.381,398.650,-102.896,176.714,29.293,155.058
C05273=1081.374,398.412,-102.858,176.710,29.285,155.056
C05274=1081.368,398.176,-102.820,176.706,29.277,155.055
C05275=1081.362,397.938,-102.780,176.702,29.270,155.053
C05276=1081.356,397.700,-102.742,176.699,29.262,155.052
C05277=1081.349,397.454,-102.703,176.695,29.254,155.050
C05278=1081.342,397.208,-102.662,176.691,29.246,155.048
C05279=1081.336,396.961,-102.622,176.687,29.238,155.047
C05280=1081.330,396.715,-102.582,176.683,29.229,155.045
C05281=1081.323,396.468,-102.543,176.679,29.221,155.043
C05282=1081.316,396.221,-102.503,176.676,29.213,155.042
C05283=1081.309,395.974,-102.463,176.672,29.205,155.040
C05284=1081.303,395.727,-102.423,176.668,29.197,155.038
C05285=1081.297,395.481,-102.383,176.664,29.189,155.037
C05286=1081.290,395.234,-102.344,176.660,29.181,155.035
C05287=1081.284,394.987,-102.304,176.657,29.173,155.034
C05288=1081.277,394.741,-102.264,176.653,29.165,155.032
C05289=1081.271,394.494,-102.225,176.649,29.158,155.031
C05290=1081.264,394.247,-102.185,176.645,29.150,155.029
C05291=1081.258,394.000,-102.146,176.641,29.142,155.027
C05292=1081.251,393.754,-102.106,176.637,29.134,155.026
C05293=1081.245,393.507,-102.067,176.633,29.126,155.024
C05294=1081.238,393.261,-102.027,176.629,29.118,155.023
C05295=1081.232,393.014,-101.988,176.627,29.111,155.021
C05296=1081.225,392.767,-101.947,176.623,29.103,155.020
C05297=1081.218,392.520,-101.909,176.619,29.095,155.018
C05298=1081.212,392.273,-101.869,176.615,29.088,155.016
C05299=1081.205,392.027,-101.830,176.611,29.080,155.015
C05300=1081.200,391.780,-101.791,176.607,29.072,155.013
C05301=1081.193,391.534,-101.752,176.603,29.064,155.012
C05302=1081.187,391.287,-101.712,176.600,29.057,155.010
C05303=1081.180,391.040,-101.673,176.596,29.049,155.009
C05304=1081.173,390.793,-101.634,176.592,29.041,155.007
C05305=1081.167,390.546,-101.594,176.588,29.034,155.006
C05306=1081.160,390.299,-101.556,176.584,29.026,155.004
C05307=1081.153,390.053,-101.516,176.580,29.019,155.003
C05308=1081.147,389.806,-101.477,176.577,29.012,155.001
C05309=1081.140,389.559,-101.438,176.573,29.004,155.000
C05310=1081.133,389.312,-101.399,176.569,28.997,154.998
C05311=1081.128,389.066,-101.360,176.566,28.989,154.997
C05312=1081.121,388.819,-101.321,176.562,28.982,154.995
C05313=1081.114,388.572,-101.282,176.559,28.975,154.994
C05314=1081.108,388.325,-101.243,176.555,28.967,154.992
C05315=1081.101,388.078,-101.204,176.551,28.960,154.991
C05316=1081.095,387.832,-101.165,176.547,28.952,154.990
C05317=1081.088,387.586,-101.127,176.543,28.945,154.988
C05318=1081.082,387.338,-101.087,176.540,28.938,154.987
C05319=1081.075,387.092,-101.048,176.536,28.930,154.985
C05320=1081.069,386.845,-101.010,176.532,28.923,154.984
C05321=1081.063,386.598,-100.972,176.528,28.915,154.982
C05322=1081.057,386.351,-100.932,176.525,28.908,154.981
C05323=1081.050,386.105,-100.894,176.521,28.901,154.980
C05324=1081.044,385.858,-100.855,176.517,28.894,154.978
C05325=1081.033,385.459,-100.793,176.512,28.882,154.976
C05326=1081.023,385.061,-100.730,176.506,28.870,154.974
C05327=1081.013,384.664,-100.668,176.499,28.859,154.971
C05328=1081.003,384.265,-100.606,176.494,28.848,154.969
C05329=1080.996,384.018,-100.567,176.490,28.840,154.968
C05330=1080.990,383.771,-100.529,176.486,28.833,154.966
C05331=1080.984,383.524,-100.490,176.483,28.827,154.965
C05332=1080.977,383.276,-100.452,176.479,28.819,154.964
C05333=1080.971,383.030,-100.413,176.475,28.812,154.962
C05334=1080.965,382.783,-100.375,176.472,28.805,154.961
C05335=1080.958,382.537,-100.337,176.468,28.798,154.960
C05336=1080.952,382.289,-100.299,176.464,28.791,154.958
C05337=1080.946,382.043,-100.260,176.461,28.784,154.957
C05338=1080.939,381.796,-100.222,176.457,28.777,154.955
C05339=1080.933,381.548,-100.184,176.453,28.770,154.954
C05340=1080.926,381.302,-100.145,176.451,28.763,154.953
C05341=1080.920,381.055,-100.107,176.447,28.756,154.951
C05342=1080.914,380.808,-100.069,176.443,28.750,154.950
C05343=1080.907,380.561,-100.031,176.440,28.743,154.949
C05344=1080.901,380.314,-99.993,176.436,28.736,154.947
C05345=1080.895,380.067,-99.955,176.432,28.729,154.946
C05346=1080.889,379.820,-99.917,176.429,28.722,154.945
C05347=1080.881,379.574,-99.879,176.425,28.715,154.944
C05348=1080.875,379.326,-99.841,176.422,28.709,154.942
C05349=1080.869,379.079,-99.803,176.418,28.702,154.941
C05350=1080.862,378.832,-99.765,176.414,28.695,154.940
C05351=1080.857,378.585,-99.727,176.411,28.688,154.938
C05352=1080.851,378.339,-99.689,176.407,28.681,154.937
C05353=1080.844,378.091,-99.651,176.404,28.675,154.936
C05354=1080.837,377.845,-99.613,176.400,28.669,154.935
C05355=1080.831,377.598,-99.575,176.396,28.662,154.933
C05356=1080.825,377.351,-99.537,176.393,28.655,154.932
C05357=1080.818,377.104,-99.499,176.389,28.648,154.931
C05358=1080.812,376.857,-99.462,176.386,28.642,154.929
C05359=1080.806,376.610,-99.425,176.382,28.635,154.928
C05360=1080.800,376.362,-99.387,176.379,28.628,154.927
C05361=1080.794,376.116,-99.349,176.375,28.622,154.926
C05362=1080.787,375.868,-99.311,176.371,28.615,154.924
C05363=1080.781,375.621,-99.273,176.368,28.609,154.923
C05364=1080.775,375.375,-99.236,176.364,28.602,154.922
C05365=1080.768,375.128,-99.198,176.361,28.596,154.921
C05366=1080.762,374.881,-99.160,176.357,28.589,154.919
C05367=1080.757,374.633,-99.123,176.354,28.582,154.918
C05368=1080.749,374.386,-99.086,176.350,28.576,154.917
C05369=1080.743,374.140,-99.048,176.347,28.569,154.916
C05370=1080.737,373.893,-99.010,176.343,28.563,154.915
C05371=1080.731,373.645,-98.973,176.340,28.556,154.913
C05372=1080.725,373.398,-98.936,176.336,28.550,154.912
C05373=1080.719,373.152,-98.898,176.332,28.543,154.911
C05374=1080.712,372.904,-98.861,176.329,28.537,154.910
C05375=1080.706,372.657,-98.823,176.325,28.531,154.909
C05376=1080.700,372.410,-98.787,176.322,28.525,154.907
C05377=1080.693,372.163,-98.749,176.318,28.518,154.906
C05378=1080.688,371.947,-98.717,176.315,28.512,154.905
C05379=1080.683,371.731,-98.684,176.313,28.507,154.904
C05380=1080.677,371.516,-98.651,176.310,28.502,154.903
C05381=1080.671,371.300,-98.619,176.307,28.496,154.902
C05382=1080.665,371.084,-98.586,176.304,28.491,154.901
C05383=1080.660,370.868,-98.554,176.300,28.485,154.900
C05384=1080.654,370.653,-98.522,176.297,28.480,154.899
C05385=1080.649,370.436,-98.489,176.294,28.474,154.898
C05386=1080.643,370.189,-98.453,176.291,28.468,154.897
C05387=1080.637,369.943,-98.415,176.287,28.462,154.896
C05388=1080.631,369.696,-98.379,176.284,28.456,154.895
C05389=1080.623,369.448,-98.341,176.280,28.450,154.893
C05390=1080.618,369.201,-98.304,176.277,28.443,154.892
C05391=1080.611,368.954,-98.268,176.273,28.437,154.891
C05392=1080.606,368.707,-98.231,176.270,28.431,154.890
C05393=1080.599,368.460,-98.193,176.266,28.425,154.889
C05394=1080.594,368.213,-98.156,176.263,28.418,154.888
C05395=1080.587,367.965,-98.120,176.259,28.412,154.886
C05396=1080.580,367.718,-98.083,176.256,28.406,154.885
C05397=1080.574,367.471,-98.045,176.253,28.400,154.884
C05398=1080.568,367.224,-98.009,176.249,28.394,154.883
C05399=1080.563,366.977,-97.972,176.246,28.388,154.882
C05400=1080.556,366.730,-97.935,176.242,28.381,154.881
C05401=1080.550,366.483,-97.899,176.239,28.376,154.880
C05402=1080.544,366.235,-97.862,176.235,28.369,154.879
C05403=1080.538,365.988,-97.825,176.232,28.363,154.877
C05404=1080.531,365.741,-97.789,176.229,28.357,154.876
C05405=1080.525,365.493,-97.752,176.225,28.351,154.875
C05406=1080.519,365.246,-97.715,176.222,28.345,154.874
C05407=1080.513,364.999,-97.679,176.218,28.339,154.873
C05408=1080.507,364.752,-97.642,176.215,28.333,154.872
C05409=1080.501,364.505,-97.605,176.212,28.328,154.871
C05410=1080.494,364.258,-97.569,176.208,28.321,154.870
C05411=1080.488,364.011,-97.532,176.205,28.316,154.869
C05412=1080.482,363.764,-97.496,176.201,28.310,154.868
C05413=1080.475,363.517,-97.459,176.198,28.304,154.867
C05414=1080.470,363.269,-97.423,176.195,28.298,154.866
C05415=1080.464,363.021,-97.387,176.191,28.292,154.865
C05416=1080.457,362.774,-97.350,176.188,28.286,154.863
C05417=1080.451,362.527,-97.314,176.185,28.280,154.862
C05418=1080.445,362.280,-97.278,176.181,28.274,154.861
C05419=1080.439,362.033,-97.242,176.178,28.269,154.860
C05420=1080.432,361.786,-97.205,176.174,28.263,154.859
C05421=1080.426,361.539,-97.169,176.171,28.257,154.858
C05422=1080.420,361.291,-97.133,176.168,28.251,154.857
C05423=1080.414,361.044,-97.097,176.164,28.245,154.856
C05424=1080.408,360.796,-97.061,176.160,28.240,154.855
C05425=1080.401,360.549,-97.024,176.157,28.234,154.854
C05426=1080.395,360.302,-96.988,176.153,28.228,154.853
C05427=1080.390,360.054,-96.952,176.150,28.222,154.852
C05428=1080.383,359.807,-96.915,176.147,28.217,154.851
C05429=1080.377,359.559,-96.879,176.143,28.211,154.850
C05430=1080.371,359.312,-96.843,176.140,28.205,154.849
C05431=1080.364,359.065,-96.808,176.137,28.200,154.848
C05432=1080.358,358.818,-96.771,176.133,28.194,154.847
C05433=1080.352,358.570,-96.736,176.130,28.188,154.846
C05434=1080.342,358.155,-96.675,176.125,28.178,154.844
C05435=1080.331,357.740,-96.614,176.119,28.169,154.842
C05436=1080.321,357.324,-96.555,176.113,28.160,154.841
C05437=1080.311,356.909,-96.494,176.108,28.150,154.839
C05438=1080.305,356.662,-96.459,176.104,28.145,154.838
